// EVENT CODE //
	FB_AlarmCodeManager(
		bAlarm1			:= MesDataExd.AX_PowerCol[1].MesData.MesAcSwitchClosed,																							// AC Switch Closed for PCS 1
		bAlarm2			:= MesDataExd.MesData.MesOpened_Dc, 																											// DC Switch Closed
		bAlarm3			:= MesDataExd.MesData.OUT_CmdStandby, 																												// Soft stop command
		bAlarm4			:= MesDataExd.MesData.MesOnGrid,																													// OnGrid Mode is activated
		bAlarm5			:= MesDataExd.MesData.MesOffGrid, 																													// Offgrid Mode is activated
		bAlarm6			:= MesDataExd.MesData.OUT_CmdStart, 																												// Cmd Start
		bAlarm7			:= MesDataExd.MesData.OUT_CmdStop, 																												// Full stop command
		bAlarm8			:= MesDataExd.OUT_CmdBlackStart, 																											// Cmd BlackStart
		bAlarm9			:= MesDataExd.AX_PowerCol[1].MesRegAlarm2.9 OR MesDataExd.AX_PowerCol[2].MesRegAlarm2.9 OR MesDataExd.AX_PowerCol[3].MesRegAlarm2.9,			// Grid collapsed 
		bAlarm10		:= MesDataExd.AX_PowerCol[2].MesData.MesAcSwitchClosed,																							// AC Switch Closed for PCS 2
		bAlarm11		:= SEL(ParamNbPowerCol>2 ,  FALSE, MesDataExd.AX_PowerCol[3].MesData.MesAcSwitchClosed),																// AC Switch Closed for PCS 3
		bAlarm12		:= MesDataExd.MesData.MesOpened_Ac, 																											// Ac breaker is Closed. 
		bAlarm13		:= MesDataExd.MesData.MesState_Precharge,                                                                                            					// ESS - INV : Precharge
		bAlarm14		:= NOT MesDataExd.OUT_CmdGridMode,                                                                                                         // OnGrid command
		bAlarm15		:= MesDataExd.OUT_CmdGridMode, 																											// OffGrid command
		wAlarmCode		=>MesDataExd.MesData.MesEventCode);                                                                                           					// 
		

NumAlarmsActive := 0;
AX_AlarmWords := AX_AlarmWords_Null;
MesNbMots := 2;
FOR KK := 1 TO MesNbMots DO			// Combien j'ai de mots
	ID_Journal := 15 + (ParamEssNum-1) * MesNbMots * CstNbPcs_ESS_G + (ParamPcsNum - 1) * CstNbPcs_ESS_G + (KK- 1);
	FOR LL := 1 TO 15 DO 	// Les bits 
		WordTest := ROR(FUN_Alarms.AX_RecupWord[ID_Journal],LL);
		IF WordTest.0 THEN
			NumAlarmsActive := NumAlarmsActive + 1;
			AX_AlarmWords[NumAlarmsActive].Message := FUN_Alarms.AX_Journal[ID_Journal][LL].Message;
		ELSE
			AX_AlarmWords[NumAlarmsActive+1].Message := '';
		END_IF
	END_FOR
END_FOR		

NumAlarmsActiveJema := 0;
AX_AlarmWordsJema := AX_AlarmWordsJema_Null;
MesNbMots := 15;
FOR KK := 1 TO MesNbMots DO			// Combien j'ai de mots
	FOR LL := 1 TO 15 DO 	// Les bits 
		ID_Journal := 57 + (ParamEssNum-1) * MesNbMots * CstNbPcs_ESS_G + (ParamPcsNum - 1) * CstNbPcs_ESS_G + (KK- 1);
		WordTest := ROR(FUN_Alarms.AX_RecupWord[ID_Journal],LL);
		IF WordTest.0 THEN
			NumAlarmsActiveJema := NumAlarmsActiveJema + 1;
			AX_AlarmWordsJema[NumAlarmsActiveJema].Message := FUN_Alarms.AX_Journal[ID_Journal][LL].Message;
		ELSE
			AX_AlarmWordsJema[NumAlarmsActiveJema+1].Message := '';
		END_IF
	END_FOR
END_FOR
END_METHOD

METHOD M_CP
//////////////////
//  Emulator
/////////////////

VAR 
	// Method local variables (reinitialized at each cycle) 
	
END_VAR


SUPER^.M_CP() ; 




Trig_Cmd_Read(CLK:=IN_CmdToggleRead);
Trig_Cmd_Write(CLK:=IN_CmdToggleWrite);
	
IF Trig_Cmd_Read.Q THEN
	IN_CmdToggleRead := FALSE;
	MesDataExd.MesData.MesCP_Read := NOT MesDataExd.MesData.MesCP_Read;
END_IF


IF Trig_Cmd_Write.Q THEN
	IN_CmdToggleWrite := FALSE;
	MesDataExd.MesData.MesCP_Write := NOT MesDataExd.MesData.MesCP_Write;
END_IF
END_METHOD

METHOD M_Evaluate : BOOL
VAR_INPUT
END_VAR
VAR
	KK : UINT;
	bTest: BOOL;
	MesAlarmPcs: BOOL;
	AX_Journal : ARRAY[57..57] of array[1..15] of ST_ValuesAlarms;
END_VAR
// External values update :
//	DataSystemBMS 				:= AX_ESS[ParamEssNum].AX_Bat[ParamPcsNum].MesDataExd;

// Gestion des watchdogs
	Trig_Watchdog(CLK := MesHeartbeat_Old <> MesDataExd.MesData.MesHeartBeat);
	IF Trig_Watchdog.Q 	THEN
		MesHeartbeat_Old := MesDataExd.MesData.MesHeartBeat;
		MesStatusWatchdog := NOT MesStatusWatchdog;
	END_IF


// Gestion des Start/Stop par SOC Low

	TRIG_SocStop			(clk := NOT MesDataExd.MesData.MesState.0 AND NOT MesDataExd.MesData.MesState.4 AND DataSystemBMS.MesSoCConnected <= ParamSocStop);
	
	IF TRIG_SocStop.Q THEN
		MesDataExd.MesData.MesState.4 := TRUE;
	END_IF
	
	
	TRIG_SocStop_Again(CLK := Time_Discharge_LowSoc > ParamTimeLowSocToRecharge);
	IF NOT MesDataExd.MesData.MesState.0 AND MesDataExd.MesData.MesState.4 AND MesDataExd.MesData.MesPdc >= 0 THEN
		Time_Discharge_LowSoc := Time_Discharge_LowSoc + TIME() - Time_Start_Discharge_LowSoc;
	ELSIF MesDataExd.MesData.MesState.0 AND (NOT MesDataExd.MesData.MesState.4 OR Time_Discharge_LowSoc >= ParamTimeLowSocToRecharge) THEN
		Time_Discharge_LowSoc := T#0S;
	END_IF
	Time_Start_Discharge_LowSoc := TIME();
	
	TRIG_BackToNormalSoc(CLK := MesDataExd.MesData.MesState.4 AND DataSystemBMS.MesSoCConnected > ParamSocStop);
	IF TRIG_BackToNormalSoc.Q THEN
		MesDataExd.MesData.MesState.4 := 0;
	END_IF
	
	
	
	IF ParamAllowRechargeLowSoc THEN
		TRIG_Recharge_LowSoc(CLK := NOT MesDataExd.MesData.MesState.0 AND NOT MesDataExd.MesData.MesState.4 AND DataSystemBMS.MesSoCConnected <= ParamSocRecharge);
		IF TRIG_Recharge_LowSoc.Q THEN
			MesDataExd.MesData.MesState.3 := TRUE;
		END_IF
		
		TRIG_RechargeBackToNormalSoc(CLK := MesDataexd.MesData.MesState.3 AND DataSystemBMS.MesSoCConnected >= ParamSocMin_G);
		IF TRIG_RechargeBackToNormalSoc.Q THEN
			MesDataexd.MesData.MesState.3 := FALSE;
		END_IF
	END_IF
	
	
	
// PROPERTIES UPDATE // 
	// Controller
	
	MesDataExd.MesData.MesP 	:= 0 ; 
	MesDataExd.MesData.MesPdc 	:= 0 ;
	MesDataExd.MesData.MesQ 	:= 0 ; 
	MesDataExd.MesData.MesI 	:= 0 ; 			
	MesDataExd.MesData.MesIdc 	:= 0 ; 		
	MesDataExd.MesData.MesTemp	:= 0 ;
	
	MesDataExd.MesData.MesAlarmCom					:= TRUE ; 	// All PCS in Com alarm . 			
	MesDataExd.MesData.MesALOPowerCol_Connected 			:= FALSE; 	// At least one inverter connected and not in alarm			
	MesDataExd.MesData.MesFreqReg_Active 			:= FALSE;
	MesDataExd.MesData.MesUReg_Active 				:= FALSE;

	// Update PCS Values	
	FOR KK:= 1 TO ParamNbPowerCol DO 
		MesDataExd.MesData.MesP 						:= MesDataExd.AX_PowerCol[KK].MesData.MesP + MesDataExd.MesData.MesP  ; 
		MesDataExd.MesData.MesI 						:= MesDataExd.AX_PowerCol[KK].MesData.MesI + MesDataExd.MesData.MesI  ; 
		MesDataExd.MesData.MesPdc 						:= MesDataExd.AX_PowerCol[KK].MesData.MesPdc + MesDataExd.MesData.MesPdc  ; 
		MesDataExd.MesData.MesQ 						:= -MesDataExd.AX_PowerCol[KK].MesData.MesQ + MesDataExd.MesData.MesQ  ; 
		MesDataExd.MesData.MesIdc 						:= MesDataExd.AX_PowerCol[KK].MesData.MesIdc + MesDataExd.MesData.MesIdc  ; 
		MesDataExd.MesData.MesFreqReg_Active			:= MesDataExd.MesData.MesFreqReg_Active 			OR MesDataExd.AX_PowerCol[KK].MesDeratingWord.6 OR MesDataExd.AX_PowerCol[KK].MesDeratingWord.7 ;
		MesDataExd.MesData.MesUReg_Active				:= MesDataExd.MesData.MesUReg_Active 				OR MesDataExd.AX_PowerCol[KK].MesDeratingWord.4 OR MesDataExd.AX_PowerCol[KK].MesDeratingWord.5 ;
		MesAlarmPcs										:= MesDataExd.AX_PowerCol[KK].MesRegAlarm0 > 0 		OR MesDataExd.AX_PowerCol[KK].MesRegAlarm1 > 0 	OR MesDataExd.AX_PowerCol[KK].MesRegAlarm2 > 0 OR MesDataExd.AX_PowerCol[KK].MesRegAlarm3 > 0 OR MesDataExd.AX_PowerCol[KK].MesRegAlarm4 > 0;                                        	
		MesDataExd.MesData.MesAlarmCom					:= MesDataExd.MesData.MesAlarmCom 					AND AX_PcsHeartbit[KK];
		MesDataExd.MesData.MesALOPowerCol_Connected 			:= MesDataExd.MesData.MesALOPowerCol_Connected 			OR MesDataExd.AX_PowerCol[KK].MesData.MesAcSwitchClosed (*FAT TESTAND NOT MesAlarmPcs *);
	
		MesDataExd.MesData.MesTemp 						:= MesDataExd.MesData.MesTemp + MesDataExd.AX_PowerCol[KK].MesData.MesTemp/ParamNbPowerCol;
	
			
	END_FOR 
	
	MesDataExd.MesData.MesCosPhi 				:= SEL(	(MesDataExd.MesData.MesP=0) AND  (MesDataExd.MesData.MesQ =0 ), MesDataExd.MesData.MesP / SQRT(EXPT(MesDataExd.MesData.MesP, 2) + EXPT(MesDataExd.MesData.MesQ, 2))   , 1) ; 		
	MesDataExd.MesData.MesFreq					:= SEL(MesDataExd.AX_PowerCol[1].MesData.MesFreq=0 ,MesDataExd.AX_PowerCol[1].MesData.MesFreq , SEL(MesDataExd.AX_PowerCol[2].MesData.MesFreq=0 ,MesDataExd.AX_PowerCol[2].MesData.MesFreq ,MesDataExd.AX_PowerCol[3].MesData.MesFreq ))   ; 		
	MesDataExd.MesData.MesU 					:= SEL(MesDataExd.AX_PowerCol[1].MesData.MesU=0 ,MesDataExd.AX_PowerCol[1].MesData.MesU , SEL(MesDataExd.AX_PowerCol[2].MesData.MesU=0 ,MesDataExd.AX_PowerCol[2].MesData.MesU ,MesDataExd.AX_PowerCol[3].MesData.MesU ))   ; 		
	MesDataExd.MesData.MesUdc 					:= SEL(MesDataExd.AX_PowerCol[1].MesData.MesUdc=0 ,MesDataExd.AX_PowerCol[1].MesData.MesUdc , SEL(MesDataExd.AX_PowerCol[2].MesData.MesUdc=0 ,MesDataExd.AX_PowerCol[2].MesData.MesUdc ,MesDataExd.AX_PowerCol[3].MesData.MesUdc ))   ; 			
	 
	
//--------------------------------------------------------------------------------//
// 							Gestion des setpoints								  //
//--------------------------------------------------------------------------------//
	
// Gestion de la puissance dispo batterie		
	//  MesDataExd.MesData.CalDynamicEfficiencyPcs := (ParamRendementPcsNom  - ParamRendementPcsMin)* (1-EXP(-(abs.MesDataExd.MesData.CalP)/ParamPnom)*100/ParamTauxDeChargeRef)) + ParamRendementPcsMin;

// Gestion des limites hautes de SoC
	RS_hystlimitmax(SET:= DataSystemBMS.MesSoCConnected >= ParamSocMax_G , RESET1:= DataSystemBMS.MesSoCConnected < ParamSocHigh) ; 
	RS_hystlimitmin(SET:= DataSystemBMS.MesSoCConnected <= ParamSocMin_G , RESET1:= DataSystemBMS.MesSoCConnected > ParamSocLow) ; 
	
	IF DataSystemBMS.MesSoCConnected >= ParamSocHigh THEN
		CalPmaxCorr_highSoC := (ParamSocMax_G - DataSystemBMS.MesSoCConnected)/(ParamSocMax_G - ParamSocHigh );
	ELSE 
		CalPmaxCorr_highSoC := 1 ;
	END_IF 
	IF DataSystemBMS.MesSoCConnected <= ParamSocLow THEN
		CalPminCorr_lowSoC := (ParamSocMin_G - DataSystemBMS.MesSoCConnected)/(ParamSocMin_G - ParamSocLow );
	ELSE
		CalPminCorr_lowSoC := 1;
	END_IF
	
	IF (datasystembms.MesData.MesCCL <> 0 OR datasystembms.MesData.MesDCL <> 0) AND DataSystemBMS.MesUdcConnected <> 0 THEN
		MesDataExd.MesData.MesSmax_ChargeFromBat 		:=  SEL(RS_hystlimitmax.Q1, 1, 0) * CalPmaxCorr_highSoC * MIN(DataSystemBMS.MesData.MesCCL*ParamChargeEfficiency/100,	ParamPn);
		MesDataExd.MesData.MesSmax_DischargeFromBat 	:=  SEL(RS_hystlimitmin.Q1, 1, 0) * CalPminCorr_lowSoC * MIN(DataSystemBMS.MesData.MesDCL*ParamDischargeEfficiency/100,	ParamPn);
	ELSE
		MesDataExd.MesData.MesSmax_ChargeFromBat := 0;
		MesDataExd.MesData.MesSmax_DischargeFromBat := 0;
	END_IF
	

// Local
	// Si je suis en local, je désactive le micro cycling et je réecris le setpoint d'input	
		IF MesDataExd.MesData.OUT_CmdPcsLocal THEN
			IN_SetptP := IN_SetptP_Local;
			IN_SetptQ := IN_SetptQ_Local;
			IN_SetptU := IN_SetptU_Local;
			IN_SetptF := IN_SetptF_Local;
		END_IF

	MesDataExd.MesData.OUT_SetptSMax := MIN(MesDataExd.MesData.MesAvailability * MesDataExd.MesData.MesSnom/100.0,  ParamPn);

IF ParamPoverQ THEN 
	// Le setpoint Max correspond à la dispo * la puissance nominale
	MesDataExd.MesData.OUT_SetptPMax := MIN(MesDataExd.MesData.MesSmax_DischargeFromBat, MesDataExd.MesData.OUT_SetptSMax);
	MesDataExd.MesData.OUT_SetptPMin := - MIN(MesDataExd.MesData.MesSmax_ChargeFromBat, MesDataExd.MesData.OUT_SetptSMax);

	// Min
	IF ABS(MesDataExd.MesData.OUT_SetptSMax) > ABS(MesDataExd.MesData.OUT_SetptP) THEN
		MesDataExd.MesData.OUT_SetptQMax		:= MIN(ParamQn, SQRT(EXPT(MesDataExd.MesData.OUT_SetptSMax, 2) - EXPT(MesDataExd.MesData.OUT_SetptP, 2)));
	ELSE
		MesDataExd.MesData.OUT_SetptQMax := 0;
	END_IF
	IF ABS(MesDataExd.MesData.OUT_SetptSMax) > ABS(MesDataExd.MesData.OUT_SetptP) THEN
		MesDataExd.MesData.OUT_SetptQMin		:= -MIN(ParamQn,SQRT( EXPT(MesDataExd.MesData.OUT_SetptSMax, 2) - EXPT(MesDataExd.MesData.OUT_SetptP, 2)));
	ELSE 
		MesDataExd.MesData.OUT_SetptQMin := 0;
	END_IF
ELSE
	MesDataExd.MesData.OUT_SetptQMax := SEL(MesDataExd.MesData.MesP = 0, SEL(MesDataExd.MesData.MesP>0, MesDataExd.MesData.MesSmax_ChargeFromBat, MesDataExd.MesData.MesSmax_DischargeFromBat), MIN(MesDataExd.MesData.MesSmax_ChargeFromBat, MesDataExd.MesData.MesSmax_DischargeFromBat));
	MesDataExd.MesData.OUT_SetptQMin := -MesDataExd.MesData.OUT_SetptQMax;
		
	MesDataExd.MesData.OUT_SetptPMax		:= MIN(SQRT(EXPT(MesDataExd.MesData.MesSmax_ChargeFromBat, 2) - EXPT(MesDataExd.MesData.OUT_SetptQ, 2)),  SEL(DataSystemBMS.MesSoCConnected < ParamSocMin_G, ParamPn, 0));
	MesDataExd.MesData.OUT_SetptPMin		:= MAX(SQRT(EXPT(MesDataExd.MesData.MesSmax_DischargeFromBat, 2) - EXPT(MesDataExd.MesData.OUT_SetptQ, 2)),  SEL(DataSystemBMS.MesSoCConnected > ParamSocMax_G, ParamPn, 0));
END_IF

// J'affecte les variables que je vais écrire
IF MesDataExd.OUT_CmdP THEN
	IF ParamAllowRechargeLowSoc AND MesDataExd.MesData.MesState.3 THEN
		IN_SetptP := MIN(IN_SetptP, - ABS(ParamPrechargeLowSoc)) ;
	END_IF
	MesDataExd.MesData.OUT_SetptP		:= MIN(MAX(IN_SetptP, MesDataExd.MesData.OUT_SetptPMin), MesDataExd.MesData.OUT_SetptPMax);
	
ELSE
	MesDataExd.MesData.OUT_SetptP 		:= 0;
END_IF

IF MesDataExd.OUT_CmdQ THEN
	MesDataExd.MesData.OUT_SetptQ		:= -MIN(MAX(IN_SetptQ, MesDataExd.MesData.OUT_SetptQMin), MesDataExd.MesData.OUT_SetptQMax);
ELSE
	MesDataExd.MesData.OUT_SetptQ 		:= 0;
END_IF

MesDataExd.OUT_SetptV := IN_SetptU;
MesDataExd.OUT_SetptF := IN_SetptF;


TON_CmdQ_On				(IN := MesDataExd.OUT_CmdQ 						AND NOT MesDataExd.MesData.MesID_State_Inv.4, PT := ParamTimeoutCmdQ);		
TON_CmdQ_Off			(IN :=  NOT MesDataExd.OUT_CmdQ  				AND MesDataExd.MesData.MesID_State_Inv.4, PT := ParamTimeoutCmdQ);				   	
TON_CmdCosPhi_On		(IN := MesDataExd.OUT_CmdCosPhi 				AND NOT MesDataExd.MesData.MesID_State_Inv.5, PT := ParamTimeoutCmdCosPhi);		
TON_CmdCosPhi_Off		(IN :=  NOT MesDataExd.OUT_CmdCosPhi 			AND MesDataExd.MesData.MesID_State_Inv.5, PT := ParamTimeoutCmdCosPhi);		
TON_FreqReg_On			(IN := MesDataExd.OUT_CmdFreqregMode 			AND NOT MesDataExd.MesData.MesID_State_Inv.2, PT := ParamTimeoutPvF);			
TON_FreqReg_Off			(IN :=  NOT MesDataExd.OUT_CmdFreqregMode 		AND MesDataExd.MesData.MesID_State_Inv.2, PT := ParamTimeoutPvF	);		
TON_UReg_On				(IN := MesDataExd.OUT_CmdUregMode 				AND NOT MesDataExd.MesData.MesID_State_Inv.1, PT := ParamTimeoutQvU	);		
TON_UReg_Off			(IN :=  NOT MesDataExd.OUT_CmdUregMode 			AND MesDataExd.MesData.MesID_State_Inv.1, PT := ParamTimeoutQvU	);		
TON_CmdGridFormer		(IN := MesDataExd.OUT_CmdGridMode 				AND NOT MesDataExd.MesData.MesID_State_Inv.10, PT := ParamTimeoutGridFormerTransition	);		
TON_CmdGridFeeder		(IN :=  NOT MesDataExd.OUT_CmdGridMode			AND MesDataExd.MesData.MesID_State_Inv.10, PT := ParamTimeoutGridFeederTransition	);		
TON_CmdStop				(IN := MesDataExd.MesData.OUT_CmdStop					AND MesDataExd.MesData.MesState.0);
TON_CmdStart			(IN := MesDataExd.MesData.OUT_CmdStart					AND NOT MesDataExd.MesData.MesState.0);
END_METHOD

METHOD M_Init

VAR 

END_VAR
SUPER^.M_Init() ; 

MesDataExd.MesData.MesState.0 := TRUE; // Initialize state to OFF

MesDataExd.OUT_CmdP := TRUE;
MesDataExd.OUT_CmdQ := TRUE;

MesDataExd.MesData.MesCP_Read := TRUE;
MesDataExd.MesData.MesCP_Write := TRUE;
END_METHOD

METHOD M_Read
//////////////////
//  Read Modbus Variable for PCS . 
/////////////////

VAR 
	// Method local variables (reinitialized at each cycle) 
	MW 						: FB_MergeWordsToDint; 

	
	MesPsetPt_Temp 			: REAL ;
	MesQsetPt_Temp			: REAL ;
	MesPavailablePcs_Temp	: REAL;
	MesPavailable_Temp		: REAL;
	
	ComErrorPcs_Temp		: WORD;
	
	KK						: BYTE;  					// FOR Loop 
	LL						: BYTE;						// Alarm Loop

	MesPsetPtPcs_temp		: ARRAY[1..CstNbPcs_ESS_G] OF  REAL; // Setpt lu sur le module
	MesQsetPtPcs_temp		: ARRAY[1..CstNbPcs_ESS_G] OF  REAL;

	AX_Qty					: ARRAY[1..3] OF WORD := [75, 68, 68];
	AX_Addr					: ARRAY[1..3] OF WORD := [1100, 1200, 1300];
	bReadChanged : BOOL;

END_VAR


IF MesDataExd.MesData.MesCP_Read  THEN	
// MODBUS REQUEST//

		ModbusRead[4]
		(
			tTimeout		:= ParamTimeout,
			nUnitID			:= ParamUnitID,
			sIPAddr			:= ParamIPAddress ,
			ClockRead		:= ClockRead AND MesDataExd.MesData.MesCP_Read,
			nTcpPort		:= ParamTcpPort,
			nQuantity		:= 75,
			Reset			:= IN_CmdReset,
			nMBAddr			:= 1100  ,//Access every PCS power modules
			cbLength		:= SIZEOF(MesBlock1_Temp[4]) , 
			pDestAddr		:= ADR(MesBlock1_Temp[4]),
			ModbusReadAlarm	=>MesModbusReadAlarm[4]
		);
			
	bReadChanged := MEMCMP(pBuf1 := ADR(MesBlock1_Temp_Old), pBuf2 := ADR(MesBlock1_Temp), n := SIZEOF(MesBlock1_Temp))<> 0;
	
	IF bReadChanged THEN
		MEMCPY(destAddr := ADR(MesBlock1_Temp_Old), srcAddr := ADR(MesBlock1_Temp), n := SIZEOF(MesBlock1_Temp_Old));
	END_IF
	TP_ReadCompleted(IN := bReadChanged, pt := ParamClockReadTime/2, Q=>MesDataExd.MesReadCompleted);

			
	// MODBUS REQUEST//
		FOR KK:=1 TO ParamNbPowerCol DO 	
			ModbusRead[KK]
			(
				tTimeout		:= ParamTimeout,
				nUnitID			:= ParamUnitID,
				sIPAddr			:= ParamIPAddress,
				ClockRead		:= ClockRead AND MesDataExd.MesData.MesCP_Read,
				nTcpPort		:= ParamTcpPort,
				nQuantity		:= AX_Qty[KK],
				Reset			:= IN_CmdReset,
				nMBAddr			:= AX_Addr[KK] ,
				cbLength		:= SIZEOF(MesBlock1_Temp[KK]) , 
				pDestAddr		:= ADR(MesBlock1_Temp[KK]),
				ModbusReadAlarm	=>MesModbusReadAlarm[KK]
			);
		END_FOR
		
		
	// MODBUS BLOCK SEPARATION/
		// Block1 (PCS) 
		FOR KK:=1 TO ParamNbPowerCol DO 	// Value per Power Column (3 per inverter IBX3)
			// Measurements
			MW( WORD_STRONG:= MesBlock1_Temp[KK][1], SIGNED:=TRUE, FIX:=1 , SIZE:=1, VAR_OUT := MesDataExd.AX_PowerCol[KK].MesData.MesUdc); 
			MW( WORD_STRONG:= MesBlock1_Temp[KK][2], SIGNED:=TRUE, FIX:=1 , SIZE:=1, VAR_OUT := MesDataExd.AX_PowerCol[KK].MesData.MesIdc); //Vérifier les signes
			MW( WORD_STRONG:= MesBlock1_Temp[KK][3], SIGNED:=FALSE, FIX:=1 , SIZE:=1, VAR_OUT := MesDataExd.AX_PowerCol[KK].MesData.MesU);
			MW( WORD_STRONG:= MesBlock1_Temp[KK][6], SIGNED:=FALSE, FIX:=1 , SIZE:=1, VAR_OUT := MesDataExd.AX_PowerCol[KK].MesData.MesI1); //Vérifier les signes
			MW( WORD_STRONG:= MesBlock1_Temp[KK][7], SIGNED:=FALSE, FIX:=1 , SIZE:=1, VAR_OUT := MesDataExd.AX_PowerCol[KK].MesData.MesI2); //Vérifier les signes
			MW( WORD_STRONG:= MesBlock1_Temp[KK][8], SIGNED:=FALSE, FIX:=1 , SIZE:=1, VAR_OUT := MesDataExd.AX_PowerCol[KK].MesData.MesI3); //Vérifier les signes
			MW( WORD_STRONG:= MesBlock1_Temp[KK][9], SIGNED:=TRUE, FIX:=1 , SIZE:=1, VAR_OUT := MesDataExd.AX_PowerCol[KK].MesData.MesPdc); // Vérifier les signes
			MW( WORD_STRONG:= MesBlock1_Temp[KK][10], SIGNED:=TRUE, FIX:=1 , SIZE:=1, VAR_OUT := MesDataExd.AX_PowerCol[KK].MesData.MesP); // Vérifier les signes
			MW( WORD_STRONG:= MesBlock1_Temp[KK][11], SIGNED:=TRUE, FIX:=1 , SIZE:=1, VAR_OUT := MesDataExd.AX_PowerCol[KK].MesData.MesQ);// Vérifier les signes
			MW( WORD_STRONG:= MesBlock1_Temp[KK][12], SIGNED:=FALSE, FIX:=3 , SIZE:=1, VAR_OUT := MesDataExd.AX_PowerCol[KK].MesData.MesCosPhi);
			MW( WORD_STRONG:= MesBlock1_Temp[KK][13], SIGNED:=FALSE, FIX:=2 , SIZE:=1, VAR_OUT := MesDataExd.AX_PowerCol[KK].MesData.MesFreq);
			
			// Inputs (Temp and IO)
			MW( WORD_STRONG:= MesBlock1_Temp[KK][15], SIGNED:=TRUE, FIX:=1 , SIZE:=1, VAR_OUT := MesDataExd.AX_PowerCol[KK].MesTempControl);
			MW( WORD_STRONG:= MesBlock1_Temp[KK][18], SIGNED:=TRUE, FIX:=1 , SIZE:=1, VAR_OUT := MesDataExd.AX_PowerCol[KK].MesTempPowerUnit);
	
			// Alarms
		MesDataExd.AX_PowerCol[KK].MesRegAlarm0:=MesBlock1_Temp[KK][24];
		MesDataExd.AX_PowerCol[KK].MesRegAlarm1:=MesBlock1_Temp[KK][25];
		MesDataExd.AX_PowerCol[KK].MesRegAlarm2:=MesBlock1_Temp[KK][26];
		MesDataExd.AX_PowerCol[KK].MesRegAlarm3:=MesBlock1_Temp[KK][27];
		MesDataExd.AX_PowerCol[KK].MesRegAlarm4:=MesBlock1_Temp[KK][28];					
	
			MW( WORD_STRONG:= MesBlock1_Temp[KK][48], SIGNED:=TRUE, FIX:=1 , SIZE:=1, VAR_OUT := MesDataExd.AX_PowerCol[KK].MesTempCabinet);
			
			// States
		MesDataExd.AX_PowerCol[KK].MesData.MesAcSwitchClosed := MesBlock1_Temp[KK][61].2 ;	// AC contactor status
		MesDataExd.AX_PowerCol[KK].MesDoorOpened := NOT MesBlock1_Temp[KK][61].6; // Door : 1= Close, O= Open
		MesDataExd.AX_PowerCol[KK].MesDeratingWord := MesBlock1_Temp[KK][62] ;
			
			MW( WORD_STRONG:= MesBlock1_Temp[KK][68], SIGNED:=FALSE, FIX:=0 , SIZE:=1, VAR_OUT := MesDataExd.AX_PowerCol[KK].MesHeartbit);
			
	
		END_FOR
	
		// Inverter states (à tester)
	
	MesDataExd.MesData.MesID_State_Inv				:= MesBlock1_Temp[4][67];
	MesDataExd.MesData.MesSnom						:= MIN(WORD_TO_REAL(MesBlock1_Temp[1][69]),ParamSn);	
	MesDataExd.MesData.MesAvailability				:= WORD_TO_REAL(MesBlock1_Temp[4][70]);
		
	MW( WORD_STRONG := MesBlock1_Temp[4][71], SIZE := 1, FIX := 0, SIGNED := FALSE, VAR_OUT := MesDataExd.MesHumidity);
	MW( WORD_STRONG := MesBlock1_Temp[4][72], SIZE := 1, FIX := 1, SIGNED := TRUE, VAR_OUT := MesDataExd.MesData.MesTemp);
	MesDataExd.MesData.MesTemp 						:= WORD_TO_REAL(MesBlock1_Temp[4][72])/10;
	MesDataExd.MesData.MesState_Precharge 			:= WORD_TO_BOOL(MesBlock1_Temp[4][73]);
	MesDataExd.MesData.MesOpened_Dc					:= NOT MesBlock1_Temp[4][74].0;
	MesDataExd.MesData.MesOpened_Ac					:= NOT  MesBlock1_Temp[4][61].0;
	MesDataExd.MesState_SoCLimitReached				:= MesBlock1_Temp[4][74].2;
	MesDataExd.MesData.MesOffGrid					:= MesBlock1_Temp[4][74].3;
	MesDataExd.MesData.MesOnGrid					:= MesBlock1_Temp[4][74].4;
	MesDataExd.MesData.MesHeartBeat					:= MesBlock1_Temp[4][75];
	
	
	
	
	
END_IF
END_METHOD

METHOD M_StateManager
//////////////////
// Detect which is the state of the PCS system . 
/////////////////

VAR 
	// Method local variables (reinitialized at each cycle) 

	
	ELS: INT;
END_VAR


MesDataExd.MesData.MesState.0 	:= 0;
IF NOT MesDataExd.MesData.MesALOPowerCol_Connected OR MesDataExd.MesData.MesOpened_Ac OR  MesDataExd.MesData.MesOpened_Dc THEN 
	// OFF State :  No Charger connected or all charger in alarm
	MesDataExd.MesData.MesState.0 	:= 1 ; 
END_IF

MesDataExd.MesData.MesState.1 	:= 0 ; 
IF MesDataExd.MesData.MesOffGrid THEN
	// Feeding master
	MesDataExd.MesData.MesState.1 	:= 1 ; 
END_IF	

MesDataExd.MesData.MesState.2 	:= 0 ; 
IF MesDataExd.MesData.OUT_CmdPcsLocal THEN
	MesDataExd.MesData.MesState.2 	:= 1 ; 
END_IF




SUPER^.M_StateManager() ;
END_METHOD

METHOD M_WriteCommand
//////////////////
//  Modbus Write of the command for the PCS. 
/////////////////

VAR 
	// Method local variables (reinitialized at each cycle) 
	
	AX_Adr			: ARRAY[1..3] OF UINT := [1707	, 1802	, 	0217	];
	AX_QTY			: ARRAY[1..3] OF BYTE := [41	, 33	, 	2		];
	AX_UnitID		: ARRAY[1..3] OF BYTE := [1		, 1		, 	1		];	

	KK: INT;
	
END_VAR
TRIG_CmdP_On			(CLK := IN_CmdP_On);						
TRIG_CmdP_Off			(CLK := IN_CmdP_Off);							
TRIG_CmdQ_On			(CLK := IN_CmdQ_On);                        
TRIG_CmdQ_Off			(CLK := IN_CmdQ_Off);                      
TRIG_CmdCosPhi_On		(CLK := IN_CmdCosPhi_On);              
TRIG_CmdCosPhi_Off		(CLK := IN_CmdCosPhi_Off);            
TRIG_CmdReset			(CLK := IN_CmdReset);
TRIG_FreqReg_On			(CLK := IN_CmdFreqregOn);
TRIG_FreqReg_Off		(CLK := IN_CmdFreqregOff);
TRIG_UReg_On			(CLK := IN_CmdUregOn);			
TRIG_UReg_Off			(CLK := IN_CmdUregOff);
TRIG_CmdGridFormer		(CLK := IN_CmdGridFormer);
TRIG_CmdGridFeeder		(CLK := IN_CmdGridFeeder);
TRIG_CmdOpenAC			(CLK := IN_CmdOpenAC);
TRIG_CmdOpenDC			(CLk := IN_CmdOpenDC);
TRIG_CmdStop			(CLK := IN_CmdStop);
TRIG_CmdStandby			(CLK := (IN_CmdStandby OR TON_BatComAlarm.Q)  AND NOT TP_CmdStop.Q );
TRIG_CmdStart			(CLK := IN_CmdStart AND NOT TP_CmdStop.Q AND NOT IN_CmdStopOperation AND (NOT IN_CmdPreventStart OR MesDataExd.MesData.OUT_CmdPcsLocal));
TRIG_CmdBlackStart		(CLK := IN_CmdBlackStart);	


TP_CmdPreStop			(IN := TRIG_CmdStop.Q, 																		PT := T#1S500MS);
TP_CmdPreStart			(IN := TRIG_CmdStart.Q, 																	PT := ParamTimePulseTrig);
TP_CmdOpenAC			(IN := TRIG_CmdOpenAC.Q, 																	PT := ParamTimePulseTrig);
TP_CmdOpenDC			(IN := TRIG_CmdOpenDC.Q, 																	PT := ParamTimePulseTrig);
TP_CmdStop				(IN := F_TrigPreStop.Q, 																	PT := ParamTimePulseTrig);
TP_CmdStart				(IN := F_TrigPreStart.Q, 																	PT := ParamTimePulseTrig);
TP_CmdStandby			(IN := TRIG_CmdStop.Q OR TRIG_CmdStandby.Q OR TRIG_SocStop.Q OR TRIG_SocStop_Again.Q, 	PT := ParamTimePulseTrig);
TP_Reset				(IN := TRIG_CmdReset.Q, 																	PT := ParamTimePulseTrig);
                		
                		
F_TrigPreStart			(CLK := TP_CmdPreStart.Q);
F_TrigPreStop			(CLK := TP_CmdPreStop.Q);


IF TRIG_CmdBlackStart.Q THEN
	IN_CmdBlackStart := FALSE;
END_IF
IF TRIG_CmdStop.Q THEN
	IN_CmdStop := FALSE;
END_IF
IF TRIG_CmdStart.Q THEN
	AX_ESS[ParamEssNum].AX_BAT[ParamPcsNum].IN_CmdCloseDC := TRUE;
	IN_CmdStart := FALSE;
END_IF
IF TRIG_CmdStandby.Q THEN
	IN_CmdStandby := FALSE;
END_IF

IF TRIG_CmdReset.Q THEN
	IN_CmdReset := FALSE;
END_IF

IF TRIG_CmdP_Off.Q THEN
	MesDataExd.OUT_CmdP := FALSE;
	IN_CmdP_Off := FALSE;
END_IF

IF TRIG_CmdP_On.Q THEN
	MesDataExd.OUT_CmdP := TRUE;
	IN_CmdP_On := FALSE;
END_IF
IF TRIG_CmdQ_Off.Q OR TRIG_CmdCosPhi_On.Q THEN
	MesDataExd.OUT_CmdQ := FALSE;
	IN_CmdQ_Off := FALSE;
END_IF
IF TRIG_CmdQ_On.Q THEN
	MesDataExd.OUT_CmdQ := TRUE;
	IN_CmdQ_On := FALSE;
END_IF

IF TRIG_CmdCosPhi_Off.Q OR TRIG_CmdQ_On.Q THEN
	MesDataExd.OUT_CmdCosPhi := FALSE;
	IN_CmdCosPhi_Off := FALSE;
END_IF

IF TRIG_CmdCosPhi_On.Q THEN
	MesDataExd.OUT_CmdCosPhi := TRUE;
	MesDataExd.OUT_SetptCosPhi	:= IN_SetptCosPhi;
	IN_CmdCosPhi_On := FALSE;
END_IF

IF TRIG_FreqReg_On.Q THEN
	MesDataExd.OUT_CmdFreqregMode := TRUE;
	IN_CmdFreqregOn := FALSE;
END_IF
IF TRIG_FreqReg_Off.Q THEN
	MesDataExd.OUT_CmdFreqregMode := FALSE;
	IN_CmdFreqregOff := FALSE;
END_IF

IF TRIG_UReg_On.Q THEN
	MesDataExd.OUT_CmdUregMode := TRUE;
	IN_CmdUregOn := FALSE;
END_IF
IF TRIG_UReg_Off.Q THEN
	MesDataExd.OUT_CmdUregMode := FALSE;
	IN_CmdUregOff := FALSE;
END_IF
	
IF TRIG_CmdGridFormer.Q THEN
	MesDataExd.OUT_CmdGridMode := TRUE;
	IN_CmdGridFormer := FALSE;
END_IF 
IF TRIG_CmdGridFeeder.Q OR TRIG_CmdStop.Q THEN //Si on fait une commande stop, on passe le mode en grid feeder
	MesDataExd.OUT_CmdGridMode := FALSE;
	IN_CmdGridFeeder := FALSE;
END_IF


IF IN_CmdPcsLocal THEN
	IN_CmdPcsLocal := FALSE;
	MesDataExd.MesData.OUT_CmdPcsLocal := NOT MesDataExd.MesData.OUT_CmdPcsLocal;
END_IF

IN_CmdWatchdog := CalLocalTimeStruct.wSecond MOD 2 = 0;

MesDataExd.MesData.OUT_CmdStop 			:= TP_CmdStop.Q;
MesDataExd.MesData.OUT_CmdStart 		:= TP_CmdStart.Q;
MesDataExd.OUT_CmdBlackStart 	:= TP_CmdBlackStart.Q;
MesDataExd.MesData.OUT_CmdStandby 		:= TP_CmdStandby.Q;


Trig_Write[1](CLK := MEMCMP(pBuf1 :=ADR(AX_Cmd[1]), pBuf2 := ADR(AX_Cmd_Old[1]), n := SIZEOF(AX_CMD[1]))<>0);
Trig_Write[2](CLK := MEMCMP(pBuf1 :=ADR(AX_Cmd[2]), pBuf2 := ADR(AX_Cmd_Old[2]), n := SIZEOF(AX_CMD[2]))<>0);
Trig_Write[3](CLK := MEMCMP(pBuf1 :=ADR(AX_Cmd[3]), pBuf2 := ADR(AX_Cmd_Old[3]), n := SIZEOF(AX_CMD[3]))<>0);

IF MEMCMP(pBuf1 :=ADR(AX_Cmd[1]), pBuf2 := ADR(AX_Cmd_Old[1]), n := SIZEOF(AX_CMD[1]))<>0 THEN
	MEMCPY(destAddr := ADR(AX_Cmd_Old[1]), srcAddr := ADR(AX_Cmd[1]), n:= SIZEOF(AX_Cmd[1]));
END_IF
IF MEMCMP(pBuf1 :=ADR(AX_Cmd[2]), pBuf2 := ADR(AX_Cmd_Old[2]), n := SIZEOF(AX_CMD[2]))<>0 THEN
	MEMCPY(destAddr := ADR(AX_Cmd_Old[2]), srcAddr := ADR(AX_Cmd[2]), n:= SIZEOF(AX_Cmd[2]));
END_IF		
IF MEMCMP(pBuf1 :=ADR(AX_Cmd[3]), pBuf2 := ADR(AX_Cmd_Old[3]), n := SIZEOF(AX_CMD[3]))<>0 THEN
	MEMCPY(destAddr := ADR(AX_Cmd_Old[3]), srcAddr := ADR(AX_Cmd[3]), n:= SIZEOF(AX_Cmd[3]));
END_IF			

	// Manouvers (41708)
		AX_Cmd[1][1].1:= IN_CmdOpenAC;
		AX_Cmd[1][1].2:= IN_CmdOpenDC;
		
	// SoC	
		AX_Cmd[1][2]  := REAL_TO_WORD(ParamFreqRegSoCmax); 
		AX_Cmd[1][3]  := REAL_TO_WORD(ParamFreqRegSoCmin); 
		AX_Cmd[1][4]  := REAL_TO_WORD(TRUNC(DataSystemBMS.MesSoCConnected));		// SoC connected 
		
		
	// Param voltage regulation (activate in Function Mode)
		// Regulation from voltage
		AX_Cmd[1][7]  := REAL_TO_WORD(ParamQfU_UDbHigh)		; 
		AX_Cmd[1][8]  := REAL_TO_WORD(ParamQfU_Umax)		  	; 
		AX_Cmd[1][9]  := REAL_TO_WORD(ParamQfU_UDbLow)	 	; 
		AX_Cmd[1][10] := REAL_TO_WORD( ParamQfU_Umin	)  		; 
		
		IF ParamNbPowerCol > 0 THEN 
			AX_Cmd[1][11]  := REAL_TO_WORD(MIN(MAX(-ParamQfU_QDbHigh*ParamNbPowerCol/ParamPn*1000.0, -1000 ), 1000))			; 
			AX_Cmd[1][12]  := REAL_TO_WORD(MIN(MAX(-ParamQfU_Qmax*ParamNbPowerCol/ParamPn*1000.0, -1000 ), 1000))			  	; 
			AX_Cmd[1][13]  := REAL_TO_WORD(MIN(MAX(-ParamQfU_QDbLow*ParamNbPowerCol/ParamPn*1000.0, -1000 ), 1000))		 	; 
			AX_Cmd[1][14]  := REAL_TO_WORD(MIN(MAX(-ParamQfU_Qmin*ParamNbPowerCol/ParamPn*1000.0, -1000 ), 1000))		  		; 
		ELSE
			AX_Cmd[1][11]  := 0 ; 
			AX_Cmd[1][12]  := 0 ; 
			AX_Cmd[1][13]  := 0 ; 
			AX_Cmd[1][14]  := 0 ; 
		END_IF

		
		
		AX_Cmd[1][15] := REAL_TO_WORD(A1_PP.ParamNominalVoltage)	; 
		AX_Cmd[1][16] := REAL_TO_WORD(A1_SUBMV.MesDataExd.MesData.MesU)	;	
		
	// Param frequency regulation 
		AX_Cmd[1][21] := REAL_TO_WORD(ParampfF_fDbHigh*100.0)		;
		AX_Cmd[1][22] := REAL_TO_WORD(ParamPfF_Fmax*100.0)		;
		AX_Cmd[1][23] := REAL_TO_WORD(ParamPfF_FDbLow*100.0)		;
		AX_Cmd[1][24] := REAL_TO_WORD(ParamPfF_Fmin*100.0)		;
		AX_Cmd[1][25] := REAL_TO_WORD(ParampfF_fDbHigh*100.0)		;
		AX_Cmd[1][26] := REAL_TO_WORD(ParamPfF_FDbLow*100.0)		;
		
		AX_Cmd[1][27] := REAL_TO_WORD(ParamPfF_FhystLow*100.0)	;
		AX_Cmd[1][28] := REAL_TO_WORD(ParamPfF_FhystHigh*100.0)	;		
		
		AX_Cmd[1][29] := REAL_TO_WORD(MIN(MAX(ParamPfF_PDbHigh/ParamPn*1000.0 , -1000 ), 1000)	)	;
		AX_Cmd[1][30] := REAL_TO_WORD(MIN(MAX(ParamPfF_Pmin/ParamPn	*1000.0, -1000 ), 1000)	)		;  
		AX_Cmd[1][31] := REAL_TO_WORD(MIN(MAX(ParamPfF_PDbLow/ParamPn*1000.0, -1000 ), 1000)	)		; 
		AX_Cmd[1][32] := REAL_TO_WORD(MIN(MAX(ParamPfF_Pmax/ParamPn*1000.0, -1000 ), 1000)		)	;  
		AX_Cmd[1][33] := REAL_TO_WORD(MIN(MAX(ParamPfF_PDbHigh/ParamPn*1000.0, -1000 ), 1000)	)		;		// P5 . 
		AX_Cmd[1][34] := REAL_TO_WORD(MIN(MAX(ParamPfF_PDbLow/ParamPn*1000.0, -1000 ), 1000)	)		; 


		AX_Cmd[1][35] := TIME_TO_WORD(ParamTimeSoCRangeReachedRmp/1000*10);				// (s) Time to go to 0 power (if SoC issue or if end of stable)
		AX_Cmd[1][37] := TIME_TO_WORD(ParamTimeEnterStblPriorRmp/1000*10);					// (s) Time to wait after entering the stable before ramping the P back to the setpoint
		AX_Cmd[1][36] := TIME_TO_WORD(ParamTimeFreqRegStbDuration/1000*10);				// (s) Time to stay in the stable area before it goes to 0
		
	// Function Mode
		AX_Cmd[1][38].0:= IN_CmdWatchdog; 							// PCS stops (hard stop) if watchdog does not change during more than 10sec
		AX_Cmd[1][38].1:= TP_Reset.Q;							// Reset
		AX_Cmd[1][38].2:= MesDataExd.OUT_CmdGridMode;	 				// To be tested
		AX_Cmd[1][38].3:= ParamSetPtModbusMode;					// Write 1 to send Setpoint via Modbus 
		AX_Cmd[1][38].4:= MesDataExd.OUT_CmdGridMode;				// Write 1 to switch to Master (to be tested)
		AX_Cmd[1][38].5:= MesDataExd.MesData.OUT_CmdStart; 				// Start: pas besoin de maintenir
		AX_Cmd[1][38].6:= MesDataExd.MesData.OUT_CmdStop; 					// Hard Stop : Open everything and stop charger .
		AX_Cmd[1][38].7:= MesDataExd.OUT_CmdP;						// P regulation enabled 
		AX_Cmd[1][38].8:= MesDataExd.OUT_CmdFreqregMode; 			// Send one to activate the Frequency regulation, to be tested
		AX_Cmd[1][38].9:= MesDataExd.OUT_CmdUregMode; 				// Send one to activate the voltage regulation, to be tested
		AX_Cmd[1][38].10:= MesDataExd.OUT_CmdQ;	 				// Q regulation enabled 
		AX_Cmd[1][38].11:= MesDataExd.OUT_CmdCosPhi;				// Cmd CosPhi ack
		AX_Cmd[1][38].12:= NOT ParamPoverQ;						// Param Q over P for Jema
		AX_Cmd[1][38].13:= ParamLVRT_Enabled;					// Param LVRT enable
		AX_Cmd[1][38].14:= ParamAntiIslanding_Enabled;			// Param Anti Islanding enable
		AX_Cmd[1][38].15:= MesDataExd.MesData.OUT_CmdStandby;				// Cmd Standby
		
		
	// Param Frequency regulation (2)
		AX_Cmd[1][39] := REAL_TO_WORD(DataSystemBMS.MesData.MesUdc);
	 
		AX_Cmd[1][40] := BOOL_TO_WORD(ParamDeactivateWatchdog);
	
		AX_Cmd[1][41].0 := NOT MesDataExd.OUT_CmdGridMode;
		
	// Setpoints

		AX_Cmd[2][1] := REAL_TO_WORD(MesDataExd.MesData.OUT_SetptP);					// Setpoint active power in kW
		AX_Cmd[2][2] := REAL_TO_WORD(MesDataExd.MesData.OUT_SetptQ);					// Setpoint reactive power in kVar
		AX_Cmd[2][4] := REAL_TO_WORD(MesDataExd.OUT_SetptCosPhi*1000);			// Setpoint CosPhi
		
	
//MesBatInit := DataSystemBMS.		

		AX_Cmd[2][18] := REAL_TO_WORD(DataSystemBMS.MesData.MesSoH);
		AX_Cmd[2][19] := REAL_TO_WORD(DataSystemBMS.MesUdcMin*1000);
		AX_Cmd[2][22] := REAL_TO_WORD(DataSystemBMS.MesUdcMax*1000);
		AX_Cmd[2][25] := UINT_TO_WORD(DataSystemBMS.MesNbRackConnected);
		AX_Cmd[2][26] := UINT_TO_WORD(DataSystemBMS.MesNbRackTot);
		AX_Cmd[2][28] := REAL_TO_WORD(DataSystemBMS.MesData.MesIdc*10);

		
		AX_Cmd[3][1] := REAL_TO_WORD(MesDataExd.OUT_SetptV);
		AX_Cmd[3][2] := REAL_TO_WORD(MesDataExd.OUT_SetptF*100);
		AX_Cmd[3][3] := REAL_TO_WORD(ParamFLow_droop*100);
		AX_Cmd[3][4] := REAL_TO_WORD(ParamFHigh_droop*100);
		AX_Cmd[3][5] := REAL_TO_WORD(ParamULow_droop); 
		AX_Cmd[3][6] := REAL_TO_WORD(ParamUHigh_droop);
		
		
// WRITE COMMAND //
	FOR KK := 1 TO 3 DO
		CmdWrite[KK] := ClockWrite OR Trig_Write[KK].Q;
	END_FOR
	
	// MODBUS REQUEST //	
		// Modbus Blocks write			
		ModbusWrite[1]
		(
			nTCPport			:= ParamTcpPort,
			pSrcAddr 			:= ADR(AX_Cmd[1]) ,
			cbLength			:= SIZEOF(AX_Cmd[1]) , 
			nQuantity 			:= AX_QTY[1],			
			Reset				:= CmdClearFault_G, 
			sIPAddr				:= ParamIPAddress , 
			nUnitID				:= ParamUnitID , 
			nMBAddr				:= AX_Adr[1] , 
			tTimeout			:= ParamTimeout ,
			WriteCmd			:= (ClockWrite OR Trig_Write[2].Q) AND MesDataExd.Mesdata.MesCP_Write , 
			ModbusWriteAlarm	=> MesModbusWriteCmdAlarm[1] , 
			ErrorId				=> MesModbusWriteCode[1]
		);   
			
		// Modbus Blocks write			
		ModbusWrite[2]
		(
			nTCPport			:= ParamTcpPort,
			pSrcAddr 			:= ADR(AX_Cmd[2]) ,
			cbLength			:= SIZEOF(AX_Cmd[2]) , 
			nQuantity 			:= AX_QTY[2],			
			Reset				:= CmdClearFault_G, 
			sIPAddr				:= ParamIPAddress , 
			nUnitID				:= ParamUnitID , 
			nMBAddr				:= AX_Adr[2] , 
			tTimeout			:= ParamTimeout ,
			WriteCmd			:= (ClockWrite OR Trig_Write[2].Q)  AND MesDataExd.Mesdata.MesCP_Write , 
			ModbusWriteAlarm	=> MesModbusWriteCmdAlarm[2] , 
			ErrorId				=> MesModbusWriteCode[2]
		);   				
		
		ModbusWrite[3]
		(
			nTCPport			:= ParamTcpPort,
			pSrcAddr 			:= ADR(AX_Cmd[3]) ,
			cbLength			:= SIZEOF(AX_Cmd[3]) , 
			nQuantity 			:= AX_QTY[3],			
			Reset				:= CmdClearFault_G, 
			sIPAddr				:= ParamIPAddress , 
			nUnitID				:= ParamUnitID, 
			nMBAddr				:= AX_Adr[3] , 
			tTimeout			:= ParamTimeout ,
			WriteCmd			:= (ClockWrite OR Trig_Write[3].Q)  AND MesDataExd.Mesdata.MesCP_Write , 
			ModbusWriteAlarm	=> MesModbusWriteCmdAlarm[3] , 
			ErrorId				=> MesModbusWriteCode[3]
		); 		
		
		
// ANALOG CMD 
OUT_SetptP_IO		:= REAL_TO_INT((32767-0)/(2*ParamPn)* MesDataExd.MesData.OUT_SetptP+32767/2) ;
OUT_SetptQ_IO		:= REAL_TO_INT((32767-0)/(2*ParamPn)* MesDataExd.MesData.OUT_SetptQ+32767/2) ;
END_METHOD

END_FUNCTION_BLOCK

// ---- 01_Equipement_Library/PCS/FB_PCS_PE.TcPOU
FUNCTION_BLOCK FB_PCS_PE EXTENDS FB_PCS_Base
//////////////////
// PLC controller . Jema Object 
//////////////////

VAR_INPUT PERSISTENT
	// Parameters of the Object
		ParamPrange							: REAL := 1559.0 ; (* (kW) Power range for scaling . *)

		ParamPn							: REAL := 1500.0;	(* (kW) Nominal power*)
		ParamPPcs						: REAL := 1265.0;
		ParamP							: REAL := 800;
		ParamQn							: REAL := 1500.0;	(* (kW) Nominal power*)
		ParamSmax							: REAL := 1500.0;	(* (kVA) Maximum apparent power of the PCS (lasts 30s)*)
		                       		
		ParamPoverQ							: BOOL := TRUE;		(* If P over Q is True, then Max setpoint for Q calculated from setpoint of P*)
    	                    			

		
 		ParamTempoStandby				: TIME	:= T#10S;	(* (s) Tempo to let time for PCS to apply a 0 setpoint before stopping . *)

     	         	    		
		ParamTimeSoCRangeReachedRmp			: TIME;				(* (ms) Time to ramp P back to the setpoint after the SoC reached its limits*)
		ParamTimeFreqRegStbDuration			: TIME;				(* (ms) Time to wait after entering the stable before ramping the P back to the setpoint *)
		ParamTimeStblRmp					: TIME; 			(* (ms) Time to ramp P back to the setpoint after entering the stable *)
		    
    {attribute 'OPC.UA.DA' := '1'}                		
		ParamAllowRechargeLowSoc			: BOOL := TRUE;		(* (NA) if true, the PCS will charge when SoC between Soc_Min and Soc_Stop*)
    {attribute 'OPC.UA.DA' := '1'}                		
		ParamPrechargeLowSoc				: REAL := 30;		(* (kW) setpoint sent at low SoC*)
    {attribute 'OPC.UA.DA' := '1'}                		
		ParamTimeLowSocToRecharge			: TIME := T#5M;		(* (ms) Time elapsed in low soc area before a soft stop is sent again *)

		ParamDeactivateWatchdog				: BOOL := TRUE;				(* Parameter to deactivate the watchdog*)

    {attribute 'OPC.UA.DA' := '1'}                		
		ParamSocLow							: REAL := 10;		(* (%) SoC from which we start limiting the maximal output Power*)
    {attribute 'OPC.UA.DA' := '1'}                		
		ParamSocHigh						: REAL := 85;		(* (%) SoC from which we start limiting the minimal output Power*)
    {attribute 'OPC.UA.DA' := '1'}                		
		ParamSocMin_G						: REAL := 5;		(* (%) Minimal SoC *)	
    {attribute 'OPC.UA.DA' := '1'}                		
		ParamSocMax_G						: REAL := 90;		(* (%) Maximal SoC *)	
    {attribute 'OPC.UA.DA' := '1'}                		
		ParamVdcStop						: REAL := 2.65;		(* (V) Vdcmin from which we stop the PCS*)
    {attribute 'OPC.UA.DA' := '1'}                		
		ParamVdcRecharge					: REAL := 2.68;		(* (V) Vdcmin from which we force the recharge*)
    {attribute 'OPC.UA.DA' := '1'}
		ParamVdcRechargeOK					: REAL := 2.7;		(* (V) Vdcmin from which we force the recharge*)
    {attribute 'OPC.UA.DA' := '1'}
		ParamVdcMin							: REAL := 1100;		(* (V) Vdcmin when we stop the forced recharge*)
    {attribute 'OPC.UA.DA' := '1'}
		ParamVdcLow							: REAL := 1150;		(* (V) VdcLow*)
    {attribute 'OPC.UA.DA' := '1'}
		ParamVdcMax							: REAL := 1300;		(* (V) VdcMax *)
    {attribute 'OPC.UA.DA' := '1'}
		ParamVdcHigh						: REAL := 1280;		(* (V) VdcHigh*)
    {attribute 'OPC.UA.DA' := '1'}
		ParamSocRecharge					: REAL := 4;		(* (%) SoC from which we recharge the PCS*)	
    {attribute 'OPC.UA.DA' := '1'}                		
		ParamSocRecharged					: REAL :=ParamSocMin_G+0.02*ParamSocMin_G;	(*(%) Soc from which we stop recharging the PCS*)
	{attribute 'OPC.UA.DA' := '1'}
		ParamPCharge						: REAL := -10;		(* (kW) power at which we consider the PCS Recharges*)
	{attribute 'OPC.UA.DA' := '1'}
		ParamChargeEfficiency				: REAL := 97;		(* (%) percentage of efficiency of PCS during charge*)
    {attribute 'OPC.UA.DA' := '1'}                		
		ParamDischargeEfficiency			: REAL := 97;		(* (%) percentage of efficiency of PCS during discharge*)
		
		ParamNbDU							: BYTE:=10 ; 			(* (NA) Total Number of disconnecting units (cables wired on the PCS)				*)
		ParamNbDU_PowerCol					: ARRAY[1..3] OF BYTE := [5,5,5]; (* (NA ) Number of disconnecting uits for each Power Columns *)
 		ParamSetpt_PCS_Discharge			:REAL;				(*SetptP parameter for the PCS discharge, if not given, it is equal to Pnom/4*)
		ParamSetpt_PCS_Charge				:REAL;  			(*SetptP parameter for the PCS charge, it is equol to 0.2*Pnom*)
		CP_PCSStop							:BOOL;
		CP_PCSStart							:BOOL;
		ParamSocStop						:REAL;
	     			
END_VAR 
VAR_INPUT   	                   			
	// Commands :

		IN_CmdPcsInLocalMode				: BOOL;				// PCS is not included in available PCS' pool (excluded from HPP control). 
		IN_CmdStopOperation					: BOOL;				// BESS Specific command : Stop operation		
		IN_CmdPreventStart					: BOOL;				// BESS Specific command : Prevent start	



		
		IN_CmdWatchdog						: BOOL ; 			// Activate or Deactivate the Watchdog function
	         
		IN_SetptCCLBat1						: REAL ; // (A) Maximal Charging Current For DC Input 1 
		IN_SetptCCLBat2						: REAL ; // (A) Maximal Charging Current For DC Input 2 
		IN_SetptCCLBat3						: REAL ; // (A) Maximal Charging Current For DC Input 3      
		IN_SetptDCLBat1						: REAL ; // (A) Maximal Discharging Current For DC Input 1 
		IN_SetptDCLBat2						: REAL ; // (A) Maximal Discharging Current For DC Input 2 
		IN_SetptDCLBat3						: REAL ; // (A) Maximal Discharging Current For DC Input 3      
		
		IN_CmdDisableCharge					: BOOL ; // Disable Charge ( SoC High reached )
		IN_CmdDisableDischarge				: BOOL ; // Disable Discharge ( SoC Low reached )
		IN_CmdLocalSocCalibration				: BOOL ; (*Launch Soc Calibration locally without needing the EMS*)
		IN_CmdEmsSocCalibration				: BOOL ; (*Launch Soc Calibration after EMS' orders*)
		IN_CmdTransfoSurcharge				: BOOL ;
		 
		IN_BMS_Selected						: WORD := 3;
		ParamDiff							:REAL;  	
		MesDataExd								: PCS_PE ;	
END_VAR
VAR_OUTPUT
	//Child objects
		OUT_SetptP_IO					: INT;			// (NA) Analogical value for the active power setpoint (based on ParamPnom)
		OUT_SetptQ_IO					: INT;			// (NA) Analogical value for the reactive power setpoint (based on ParamQnom)
END_VAR
VAR          



                           	
	//M_ALARMMANAGEMENT VARIABLES//  
		AX_AlarmWords						: ARRAY[1..30] OF ST_ValuesAlarms;
		AX_AlarmWords_Null					: ARRAY[1..30] OF ST_ValuesAlarms;
		AX_AlarmWordsJema					: ARRAY[1..225] OF ST_ValuesAlarms;
		AX_AlarmWordsJema_Null				: ARRAY[1..225] OF ST_ValuesAlarms;
		NumAlarmsActive						: UINT;
		NumAlarmsActiveJema					: UINT;
	//M_READ VARIABLES//            		
		FB_ModbusRead	          	: ARRAY[1..8] OF FB_ModbusRead; // (NA) FB for Modbus Reading
		AX_ModbusReadAlarm			: ARRAY[1..8] OF BOOL;
		AX_ModbusReadAlarmId		: ARRAY[1..8] OF UDINT;	
		
		FB_ModbusRead_PowerCol		: ARRAY[1.. CstNbPowerCol_PCS_G] OF FB_ModbusRead; 
		AX_ModbusReadAlarmPowerCol	: ARRAY[1.. CstNbPowerCol_PCS_G] OF BOOL;
		AX_ModbusReadAlarmIdPowerCol: ARRAY[1.. CstNbPowerCol_PCS_G] OF UDINT ;
		
		FB_ModbusWrite				: ARRAY[1..10]  OF FB_ModbusWrite;
		AX_ModbusWriteAlarm			: ARRAY[1..10]  OF BOOL;
		AX_ModbusWriteAlarmId		: ARRAY[1..10]  OF UDINT;	

		FB_ModbusRead_DU			: ARRAY[1..CstNbDU_PCS] OF FB_ModbusRead;
		AX_ModbusReadAlarmDU		: ARRAY[1.. CstNbDU_PCS] OF BOOL;
		AX_ModbusReadAlarmIDU		: ARRAY[1.. CstNbDU_PCS] OF UDINT ;	
	
		MesBlock_Temp_1 			: ARRAY [1..120] OF WORD ; 		// (NA) Temporary Block with multiple modbus reading 
		MesBlock_Temp_2 			: ARRAY [1..120] OF WORD ; 		// (NA) Temporary Block with multiple modbus reading 
		MesBlock_Temp_3 			: ARRAY [1..120] OF WORD ; 		// (NA) Temporary Block with multiple modbus reading 
		MesBlock_Temp_4 			: ARRAY [1..120] OF WORD ; 		// (NA) Temporary Block with multiple modbus reading 
		MesBlock_Temp_5 			: ARRAY[1..6] OF ARRAY [1..120] OF WORD ; 		// (NA) Temporary Block with multiple modbus reading 
		MesBlock_Temp_6 			: ARRAY[1..CstNbDU_PCS] OF ARRAY [1..6] OF WORD ; 		// (NA) Temporary Block with multiple modbus reading 
		MesBlock_Temp_7				: ARRAY [1..120] OF WORD ; 		// (NA) Temporary Block with multiple modbus reading 
		MesBlock_Temp_8				: ARRAY [0..120] OF BOOL ;

		
		MesBlockWrite1_Temp 			: WORD;							// (NA) Temporary Block with multiple modbus writing (Caution : Double Word variables)
		MesBlockWrite1_Temp_Old 		: WORD;							// (NA) Temporary Block with multiple modbus writing (Caution : Double Word variables)
		MesBlockWrite2_Temp				: ARRAY[1..3]    OF WORD;		// (NA) Temporary Block with multiple modbus writing (Caution : Double Word variables)
		MesBlockWrite2_Temp_Old			: ARRAY[1..3]    OF WORD;		// (NA) Temporary Block with multiple modbus writing (Caution : Double Word variables)
		MesBlockWrite3_Temp				: WORD;							// (NA) Temporary Block with multiple modbus writing (Caution : Double Word variables)
		MesBlockWrite3_Temp_Old			: WORD;							// (NA) Temporary Block with multiple modbus writing (Caution : Double Word variables)
		MesBlockWrite4_Temp				: WORD;		// (NA) Temporary Block with multiple modbus writing (Caution : Double Word variables)
		MesBlockWrite4_Temp_Old			: WORD;		// (NA) Temporary Block with multiple modbus writing (Caution : Double Word variables)
		MesBlockWrite5_Temp				: ARRAY[1..2]   OF WORD;		// (NA) Temporary Block with multiple modbus writing (Caution : Double Word variables)
		MesBlockWrite5_Temp_Old			: ARRAY[1..2]   OF WORD;		// (NA) Temporary Block with multiple modbus writing (Caution : Double Word variables)
		MesBlockWrite6_Temp				: ARRAY[1..6]   OF WORD;		// (NA) Temporary Block with multiple modbus writing (Caution : Double Word variables)
		MesBlockWrite6_Temp_Old			: ARRAY[1..6]   OF WORD;		// (NA) Temporary Block with multiple modbus writing (Caution : Double Word variables)
		MesBlockWrite7_Temp				: ARRAY[1..1]   OF WORD;		// (NA) Temporary Block with multiple modbus writing (Caution : Double Word variables)
		MesBlockWrite7_Temp_Old			: ARRAY[1..1]   OF WORD;		// (NA) Temporary Block with multiple modbus writing (Caution : Double Word variables)
		MesBlockWrite8_Temp				: BOOL ;
		MesBlockWrite9_Temp				: WORD;
		MesBlockWrite10_Temp			: WORD;
		TRIG_Write						: ARRAY[1..3] OF R_TRIG;

		AX_PcsHeartbit					: ARRAY [1..4] OF BOOL;
		                                
		TON_AlarmPcs					: ARRAY [1..CstNbPowerCol_PCS_G] OF TON ; 			// DesInhibate undervoltage alarms on PCS few seconds after PCS connected .  
                                    	                          	                                     
	                                    
		FB_SplitWordToByte				: FB_SplitWordToByte ; 			
                                        
	// M_EVALUATE VARIABLES//           
		MesStatusWatchdog					: BOOL;
		MesHeartbeat_Old					: WORD;
		Trig_Watchdog						: R_TRIG;
		Time_Discharge_LowSoc				: TIME;
		Time_Start_Discharge_LowSoc			: TIME;
		DataSystemBMS1						: BAT_SAFT;
		DataSystemBMS2						: BAT_SAFT;
		
	// Microcycling //
		MesMicroCyclingP					: REAL;				// (kW) Actual P for microcyling mode (if micro act = either ParamPmicro/-ParamPmicor, else 0)		
		MesMicroCyclingP_Old				: REAL;				// (kW) Active power the PCS will have during microcyling
	    MesMicroCyclingAllowed				: BOOL;				// (NA) If SoC is in range for microCycling                        		
		Trig_MicroCyclingNoLongerAllowed	: F_TRIG;			// Trig to detect falling edge of microcylingAllowed

	//M_WRITECOMMAND VARIABLES//    		
		TRIG_CmdOpenAC						: R_TRIG;										// Trig to detect an order to change Mode
		TRIG_CmdOpenDC						: R_TRIG;										// Trig to detect an order to change Mode
		TRIG_CmdReset						: R_TRIG;		

		TRIG_CmdStop						: R_TRIG;
		TRIG_CmdStandby						: R_TRIG;
		TRIG_CmdStart						: R_TRIG;
		TRIG_CmdPcsLocal					: R_TRIG;
		TRIG_LowLowSoC						: R_TRIG;
		TRIG_WriteToChangeModule			: R_TRIG;
		TRIG_ReadModule						: F_TRIG;
		CTU_ModuleNumber					: CTU;		
                            		
		TP_CmdBlackStart					: TP;				// TP To ensure R trig is detected
		TP_Reset							: TP ; 				// (NA) Maintain Reset command for a certain time 
		TP_CmdStandby						: TP;				// TP To maintain a soft stop order
		TP_Cmd_alarm						: TP;
		TP_CmdStandbyNow					: TP;
		TP_CmdStandbyRackEND				: TP;
		TP_Start							: TP;
		TRIG_StandbyNow						: R_TRIG;
		TRIG_StandbyRack					: R_TRIG;
		TRIG_StandbyRackEND					: R_TRIG;
		F_TRIG_StandbyRack					: F_TRIG;
		F_TRIG_END							: F_TRIG;
		F_TRIG_StandbyRackEND				: F_TRIG;
		TP_CmdStandbyRack					: TP;
		TRIG_Recharge_LowSoc				: R_TRIG;
		TRIG_RechargeBackToNormalSoc		: R_TRIG;
		TRIG_SocStop						: R_TRIG;
		TON_SocStop							: TON;
		TRIG_SocStop_Again					: R_TRIG;
        TRIG_BackToNormalSoc				: R_TRIG;
		CmdStopOperation					: BOOL;
		CmdInAlarmBat						: BOOL;
		MesAlarmsBackToNormal				: BOOL;
		xTest								: BOOL;
		F_TRIG_AlarmBat						: F_TRIG;
		// Pour la commande start, j'envoie une consigne pour fermer les contacteurs DC des batteries
		TP_CmdOpenAC						: TP;				// TP To ensure R trig is detected
		TP_CmdOpenDC						: TP;				// TP To ensure R trig is detected

		TP_CmdStart							: TP;				// TP To ensure R trig is detected
		TP_CmdPreStart						: TP;				// TP To send a close dc breaker order before sending start order
		F_TrigPreStart						: F_TRIG;			// failing edge to detect end of TP;
		
		// Pour la commande stop, pour éviter qu'on ouvre tout d'un coup, je faire un pré stop pendant 1,5s où j'envoie un autre de standby
		TP_CmdStop							: TP;				// TP To ensure R trig is detected
		TP_CmdPreStop						: TP;				// TP to send a soft stop before sending a stop 
		F_TrigPreStop						: F_TRIG;			// failing edge to detect end of TP;
		                            	

		TON_CmdStart			    		: TON;
		TON_CmdStop	                		: TON;
		TON_CmdStandby		        		: TON;

		Trig_Local_Start				: R_Trig;
		Trig_Local_Stop					: R_Trig;
		Trig_Local_EmergencyStop		: R_Trig;
		Trig_Start						: R_Trig;
		Trig_Stop						: R_Trig;
		Trig_Reset						: R_Trig;		


		F_TRIG_Standby: F_TRIG;
		F_TRIG_alarm:F_TRIG;
		F_TRIG_SoftStop:F_TRIG;		                            		

		
	
		TP_CmdStandbyDelay					: TP ; 				// TP to delay application of standby order
		
		
		
		bMaintainStop					: BOOL;	// Allow to keep setpoint to zero after a standby order .   RS .     	

		FB_Ramp_Standby			: FB_Ramp;	// Ramp to zero after a standby order
		FB_Ramp_StandbyQ		: FB_Ramp; // Ramp to zero after a standby order
	
			
		
		RS_hystlimitmin1					: RS;
		RS_hystlimitmax1					: RS;
		RS_hystlimitmin2					: RS;
		RS_hystlimitmax2					: RS;
 		RS_hystlimitEnergyShifmin			: RS;
		RS_hystlimitEnergyShifmax			: RS;
		
		CalPmaxCorr_highSoC1				: REAL;
		CalPminCorr_lowSoC1					: REAL;
		CalPmaxCorr_highSoC2				: REAL;
		CalPminCorr_lowSoC2					: REAL;
        	
		MesRead_Module_Number				: UINT;
		StartStop_RTrig				: R_Trig;
        // M_Calibration//
		CP_Calibration_Discharge		:BOOL; 			(*Boolean that has the condition  until when we should discharge*)
		CP_Calibration_Charge			:BOOL; 			(*Boolean that has the condition  until when we should consider the PCS charged*)
		FTrig_Discharge					: F_TRIG;		(*The Ftrig discharge will detect the descendent front and gives the Q = TRUE*)
		TP_Discharge					: TP;			(*The TP is used once the signal is TRUE, the TP's output stays true for 20minutes*)
		TP_Discharge_End				: TP;			(*The TP is used to detect the end of 20 minitus and thus change to the state to go to the recharge phase*)
		TON_Timeout_Calibration			: TP;			(*Time Out if the calibration takes too much time*)
		Trig_Timeout_Calibration		: F_TRIG;		(*Triggers the time out of calibration*)
		
		//SURCHARGE Transfo 
		TP_Surcharge 						: TP;	(*Timer to count 3 hours starting S of the PCS > S of the transformer allower*)				
		FTrig_Surcharge 					: F_TRIG;	(*Descendant front to detect the end of the 3 hours*)
		TransfoDurationSurchargeEnd			: BOOL;		(* (Nan) TRUE : it's been three hours that the transfo is surcharged FALSE otherwise*)
		MesTransfoSurchargeState			: BOOL;		(* (Nan) TRUE : The transfo is surcharged, False otherwise*)
		ParamSmaxTransfo					: INT :=1600;		(*The maximum apparent power accepted by the transformer*)   

		//Rack fault//
		MesStateFaultRack					: BOOL ;                            		
END_VAR

METHOD M_AlarmManagement
//////////////////
//  PCS Alarm Management 
/////////////////

VAR 
	// Method local variables (reinitialized at each cycle) 
	FB_AlarmCodeManager : FB_AlarmCodeManager ; 
	KK					: UINT;				// For Loop
	ComWarning			: BOOL;				// Aggregated Wcommunication warning
	ComAlarm			: BOOL;				// Aggregated communication Alarm
	
	CalAlarmPcsSynthesis: BOOL;
	LL					: UINT;
	ID_Journal			: UINT;
	WordTest			: WORD;
	MesNbMots			: UINT;
END_VAR
// COMMUNICATION //
	ComWarning 				:=  AX_ModbusReadAlarm[1] OR AX_ModbusReadAlarm[2] OR AX_ModbusReadAlarm[3] OR AX_ModbusReadAlarm[4] OR AX_ModbusReadAlarm[5] OR AX_ModbusReadAlarm[6] OR AX_ModbusReadAlarm[7];		
	ComAlarm				:=  AX_ModbusReadAlarm[1] AND AX_ModbusReadAlarm[2] AND AX_ModbusReadAlarm[3] AND AX_ModbusReadAlarm[4] AND AX_ModbusReadAlarm[5] AND AX_ModbusReadAlarm[6] AND AX_ModbusReadAlarm[7] ;

	FOR KK := 1 TO CstNbPowerCol_PCS_G DO
		ComWarning 	:= ComWarning OR AX_ModbusReadAlarmPowerCol[KK];
		ComAlarm	:= ComAlarm AND AX_ModbusReadAlarmPowerCol[KK];		
	END_FOR

	
		
	TON_ComAlarm(IN:= ComAlarm , PT:= ParamTempoComAlarm, Q=>MesComAlarm) ;	
	TON_ComWarning(IN := ComWarning, PT := ParamTempoComWarning, Q => MesComWarning);

	MesDataExd.MesData.MesAlarmCom		:= MesComAlarm ; 
	MesDataExd.MesData.MesWarningCom 	:= MesComWarning ; 

// PCS ALARM INHIBITION
FOR KK := 1 TO ParamNbPowerCol DO
	TON_AlarmPcs[KK](IN:=NOT MesDataExd.MesData.MesState.0, PT:= T#5S ) ;
END_FOR	


// SYNTHESES ALARMES //
CalAlarmPcsSynthesis := FALSE ; 
FOR KK:= 1 TO ParamNbPowerCol DO  
	CalAlarmPcsSynthesis := CalAlarmPcsSynthesis OR MesDataExd.AX_PowerCol[KK].MesIDState >16 ; 
END_FOR

// AlarmCode

// Attention une alarm doit être mise en commentaire de la manière suivante (* *), l'utilisation du // pose pb sur Bazefield 	
	
	FB_AlarmCodeManager(
		bAlarm1		:= CalAlarmPcsSynthesis		,								// Power columns Alarm Synthesis, at least one alarm active on power column
		bAlarm2		:= FALSE , //
		bAlarm3		:= FALSE , //	
		bAlarm4		:= FALSE,										            //                              			    	
		bAlarm5		:= FALSE , //
		bAlarm6		:= FALSE , //                 				
		bAlarm7		:= FALSE , //
		bAlarm8 	:= FALSE , //
		bAlarm9		:= FALSE , //
		bAlarm10	:= FALSE , //
		bAlarm11	:= MesDataExd.MesData.MesAlarmCom,                                     // Communication alarm : none of the Power Columns are responding 				
		bAlarm12	:= MesDataExd.MesData.MesAlarm,                                               	//PCS Controller general Alarm		
		bAlarm13	:= FALSE,                                               	//			
		bAlarm14	:= FALSE,                                               	//		
		bAlarm15	:= FALSE,                                               	//		
		wAlarmCode	=>MesDataExd.MesData.MesAlarmCode);		                                		
		                                                                                 	
		
		
// WARNING CODE //
	FB_AlarmCodeManager(
		bAlarm1		:= MesComWarning, 																											// Communication warning : At least one of the Power Columns are not responding 
		bAlarm2		:= MesDataExd.MesData.MesWarning,																							//PCS Controller general Warning  
		bAlarm3		:= MesDataExd.MesIDState = 10  ,  																							// LVRT is running 
		bAlarm4		:= MesDataExd.MesIDState = 11,    																							// OVRT is runnning
		bAlarm5		:= FALSE , // 
		bAlarm6		:= FALSE , // 
		bAlarm7		:= FALSE , // 
		bAlarm8		:= FALSE , // 
		bAlarm9		:= FALSE , // 
		bAlarm10	:= FALSE , // 
		bAlarm11	:= FALSE , // 
		bAlarm12	:= FALSE , // 
		bAlarm13	:= FALSE,           																										//
		bAlarm14	:= FALSE,           																										//
		bAlarm15	:= FALSE,           																										//
		wAlarmCode	=>MesDataExd.MesData.MesWarningCode);
		
// EVENT CODE //
	FB_AlarmCodeManager(
		bAlarm1			:= FALSE , // 
		bAlarm2			:= MesDataExd.MesData.MesOpened_Dc, 																											// DC Switch Closed
		bAlarm3			:= MesDataExd.MesData.OUT_CmdStandby, 																												// Soft stop command
		bAlarm4			:= MesDataExd.MesData.MesOnGrid,																													// OnGrid Mode is activated
		bAlarm5			:= MesDataExd.MesData.MesOffGrid, 																													// Offgrid Mode is activated
		bAlarm6			:= MesDataExd.MesData.OUT_CmdStart, 																												// Cmd Start
		bAlarm7			:= MesDataExd.MesData.OUT_CmdStop, 																												// Full stop command
		bAlarm8			:= FALSE , // 
		bAlarm9			:= FALSE , // 
		bAlarm10		:= FALSE , // 
		bAlarm11		:= FALSE , // 
		bAlarm12		:= MesDataExd.MesData.MesOpened_Ac, 																											// Ac breaker is Closed. 
		bAlarm13		:= FALSE , //
		bAlarm14		:= FALSE , //
		bAlarm15		:= FALSE , //
		wAlarmCode		=>MesDataExd.MesData.MesEventCode);                                                                                           					// 
		

NumAlarmsActive := 0;
AX_AlarmWords := AX_AlarmWords_Null;
MesNbMots := 2;
FOR KK := 1 TO MesNbMots DO			// Combien j'ai de mots
	ID_Journal := 15 + (ParamEssNum-1) * MesNbMots * CstNbPcs_ESS_G + (ParamPcsNum - 1) * CstNbPcs_ESS_G + (KK- 1);
	FOR LL := 1 TO 15 DO 	// Les bits 
		WordTest := ROR(FUN_Alarms.AX_RecupWord[ID_Journal],LL);
		IF WordTest.0 THEN
			NumAlarmsActive := NumAlarmsActive + 1;
			AX_AlarmWords[NumAlarmsActive].Message := FUN_Alarms.AX_Journal[ID_Journal][LL].Message;
		ELSE
			AX_AlarmWords[NumAlarmsActive+1].Message := '';
		END_IF
	END_FOR
END_FOR		

NumAlarmsActiveJema := 0;
AX_AlarmWordsJema := AX_AlarmWordsJema_Null;
MesNbMots := 15;
FOR KK := 1 TO MesNbMots DO			// Combien j'ai de mots
	FOR LL := 1 TO 15 DO 	// Les bits 
		ID_Journal := 57 + (ParamEssNum-1) * MesNbMots * CstNbPcs_ESS_G + (ParamPcsNum - 1) * CstNbPcs_ESS_G + (KK- 1);
		WordTest := ROR(FUN_Alarms.AX_RecupWord[ID_Journal],LL);
		IF WordTest.0 THEN
			NumAlarmsActiveJema := NumAlarmsActiveJema + 1;
			AX_AlarmWordsJema[NumAlarmsActiveJema].Message := FUN_Alarms.AX_Journal[ID_Journal][LL].Message;
		ELSE
			AX_AlarmWordsJema[NumAlarmsActiveJema+1].Message := '';
		END_IF
	END_FOR
END_FOR
END_METHOD

METHOD M_Calibration
VAR
	KK								: INT;
END_VAR
//SOC CALIBRATION
//Process of Calibration starting, conditions found on SAFT document
MesDataExd.MesCalibrationState.0 := 1; //Calibration Started
	FOR KK:=1 TO CstNbBat_ESS_G DO
	//	CP_Calibration_Discharge := CP_Calibration_Discharge OR (AX_ESS[ParamEssNum].AX_Bat[KK].MesDataExd.MesData.MesDCL < 36 * AX_ESS[ParamEssNum].AX_Bat[KK].MesDataExd.MesNbRackConnected AND AX_ESS[ParamEssNum].AX_Bat[KK].MesDataExd.MesIDAlarm_Vendor1.12);
	END_FOR
	
	// If the condition is not met we discharge
	IF NOT(CP_Calibration_Discharge) THEN
		MesDataExd.MesData.OUT_SetptP := ParamSetpt_PCS_Discharge;
		MesDataExd.MesCalibrationState.1 := 1; //We send the setpoint to the PCS, the PCS starts discharging
	END_IF
	
	//If the condition is met we stop the discharge and change the calibration state of the pcs
	IF CP_Calibration_Discharge THEN
		MesDataExd.MesCalibrationState.2 := 1; //Discharging done and starting 20min hold
	END_IF
	//By changing the calibration state of the PCS we can start holding off the PCS for 20min
	IF MesDataExd.MesCalibrationState.2 THEN
		TP_Discharge(IN:=MesDataExd.MesCalibrationState.2,PT:=T#20M);
		MesDataExd.MesData.OUT_SetptP := 0;
	END_IF
	
	//Once the 20min is done, we can start charging
	FTrig_Discharge(CLK := TP_Discharge.Q);
	
	IF FTrig_Discharge.Q THEN
		MesDataExd.MesCalibrationState.3 := 1;
	END_IF
	IF MesDataExd.MesCalibrationState.3 THEN
		FOR KK:=1 TO CstNbBat_ESS_G DO
				CP_Calibration_Charge := CP_Calibration_Charge AND (AX_ESS[ParamEssNum].AX_Bat[KK].MesDataExd.MesData.MesSoC >= ParamSocRecharged);
		END_FOR
		IF NOT(CP_Calibration_Charge) THEN
			 //Charging had started
			MesDataExd.MesData.OUT_SetptP := ParamSetpt_PCS_Charge;
		END_IF
		IF CP_Calibration_Charge THEN
			MesDataExd.MesCalibrationState:=0;
		END_IF
	END_IF
END_METHOD

METHOD M_CP
//////////////////
//  Emulator
/////////////////

VAR 
	// Method local variables (reinitialized at each cycle) 
	
END_VAR
	CalCP_Stop 					:=  TRUE;
	CalCP_Start					:=  NOT MesDataExd.MesData.MesAlarmCode.0 AND NOT CmdClearFault_G AND MesDataExd.MesData.MesState.0 AND  (MesDataExd.MesIDState = 2 OR MesDataExd.MesIDState = 4)AND NOT TP_CmdStop.Q AND NOT IN_CmdStopOperation AND NOT IN_CmdPreventStart ;
	
	CalCP_Reset 				:=  TRUE;
	CalCP_Standby				:= NOT TP_CmdStop.Q  ; 



SUPER^.M_CP() ; 




Trig_Cmd_Read(CLK:=IN_CmdToggleRead);
Trig_Cmd_Write(CLK:=IN_CmdToggleWrite);
	
IF Trig_Cmd_Read.Q THEN
	IN_CmdToggleRead := FALSE;
	MesDataExd.MesData.MesCP_Read := NOT MesDataExd.MesData.MesCP_Read;
END_IF


IF Trig_Cmd_Write.Q THEN
	IN_CmdToggleWrite := FALSE;
	MesDataExd.MesData.MesCP_Write := NOT MesDataExd.MesData.MesCP_Write;
END_IF
END_METHOD

METHOD M_Evaluate : BOOL
VAR_INPUT
END_VAR
VAR
	KK : UINT;
	bTest: BOOL;
	MesAlarmPcs: BOOL;
	AX_Journal : ARRAY[57..57] OF ARRAY[1..15] OF ST_ValuesAlarms;
	CalCoeffSoC_Charge			: USINT;
	CalCoeffSoC_Discharge		: USINT;
	
	DataSystemBMS		: BAT_SAFT ; 
END_VAR
// External values update :
	DataSystemBMS1 				:= AX_ESS[ParamEssNum].AX_Bat[1].MesDataExd;
	DataSystemBMS2 				:= AX_ESS[ParamEssNum].AX_Bat[2].MesDataExd;


// Gestion des Start/Stop par SOC Low
	CP_PCSStop := (DataSystemBMS1.MesData.MesUdcMin_Cell <= ParamVdcStop) OR (DataSystemBMS2.MesData.MesUdcMin_Cell <= ParamVdcStop);
	TRIG_SocStop(clk := NOT MesDataExd.MesData.MesState.0 AND NOT MesDataExd.MesData.MesState.14 AND CP_PCSStop);
	IF TRIG_SocStop.Q THEN 
		MesDataExd.MesData.MesState.14 := TRUE;
	END_IF
	
	
	TRIG_SocStop_Again(CLK := Time_Discharge_LowSoc > ParamTimeLowSocToRecharge);
	IF NOT MesDataExd.MesData.MesState.0 AND MesDataExd.MesData.MesState.14 AND MesDataExd.MesData.MesPdc >= 0 THEN
		Time_Discharge_LowSoc := Time_Discharge_LowSoc + TIME() - Time_Start_Discharge_LowSoc;
	ELSIF MesDataExd.MesData.MesState.0 AND (NOT MesDataExd.MesData.MesState.14 OR Time_Discharge_LowSoc >= ParamTimeLowSocToRecharge) THEN
		Time_Discharge_LowSoc := T#0S;
	END_IF
	Time_Start_Discharge_LowSoc := TIME();
	CP_PCSStart := (DataSystemBMS1.MesData.MesUdcMin_Cell > ParamVdcStop) OR (DataSystemBMS2.MesData.MesUdcMin_Cell > ParamVdcStop);
	TRIG_BackToNormalSoc(CLK := MesDataExd.MesData.MesState.14 AND CP_PCSStart);
	IF TRIG_BackToNormalSoc.Q THEN
		MesDataExd.MesData.MesState.14 := 0;
	END_IF
	
	
	
	IF ParamAllowRechargeLowSoc THEN
		TRIG_Recharge_LowSoc(CLK := NOT MesDataExd.MesData.MesState.0 AND NOT MesDataExd.MesData.MesState.14 AND (DataSystemBMS1.MesData.MesUdcMin_Cell <= ParamVdcRecharge OR DataSystemBMS2.MesData.MesUdcMin_Cell <= ParamVdcRecharge));
		IF TRIG_Recharge_LowSoc.Q THEN
			MesDataExd.MesData.MesState.13 := TRUE;
		END_IF
		
		TRIG_RechargeBackToNormalSoc(CLK := MesDataexd.MesData.MesState.13 AND (DataSystemBMS1.MesData.MesUdcMin_Cell >= ParamVdcRechargeOK AND DataSystemBMS2.MesData.MesUdcMin_Cell >= ParamVdcRechargeOK));
		IF TRIG_RechargeBackToNormalSoc.Q THEN
			MesDataexd.MesData.MesState.13 := FALSE;
		END_IF
	END_IF
	
	
	
// PROPERTIES UPDATE // 



//--------------------------------------------------------------------------------//
// 							Gestion des setpoints								  //
//--------------------------------------------------------------------------------//

// Gestion des limites hautes de SoC
	RS_hystlimitmax1(SET:= DataSystemBMS1.MesData.MesUdc >= ParamVdcMax , RESET1:= DataSystemBMS1.MesData.MesUdc < ParamVdcHigh) ; 
	RS_hystlimitmin1(SET:= DataSystemBMS1.MesData.MesUdc <= ParamVdcMin , RESET1:= DataSystemBMS1.MesData.MesUdc > ParamVdcLow) ; 
	RS_hystlimitmax2(SET:= DataSystemBMS2.MesData.MesUdc >= ParamVdcMax , RESET1:= DataSystemBMS2.MesData.MesUdc < ParamVdcHigh) ; 
	RS_hystlimitmin2(SET:= DataSystemBMS2.MesData.MesUdc <= ParamVdcMin , RESET1:= DataSystemBMS2.MesData.MesUdc > ParamVdcLow) ;
	
	IF DataSystemBMS1.MesData.MesUdc >= ParamVdcHigh THEN
		CalPmaxCorr_highSoC1 := (ParamVdcMax - DataSystemBMS1.MesData.MesUdc)/(ParamVdcMax - ParamVdcHigh);
	ELSE 
		CalPmaxCorr_highSoC1 := 1 ;
	END_IF
	IF DataSystemBMS2.MesData.MesUdc >= ParamVdcHigh THEN
		CalPmaxCorr_highSoC2 := (ParamVdcMax - DataSystemBMS2.MesData.MesUdc)/(ParamVdcMax - ParamVdcHigh);
	ELSE 
		CalPmaxCorr_highSoC2 := 1 ;
	END_IF
	IF DataSystemBMS1.MesData.MesUdc <= ParamVdcLow THEN
		CalPminCorr_lowSoC1 := (ParamVdcMin - DataSystemBMS1.MesData.MesUdc)/(ParamVdcMin - ParamVdcLow );
	ELSE
		CalPminCorr_lowSoC1 := 1;
	END_IF
	IF DataSystemBMS2.MesData.MesUdc <= ParamVdcLow THEN
		CalPminCorr_lowSoC2 := (ParamVdcMin - DataSystemBMS2.MesData.MesUdc)/(ParamVdcMin - ParamVdcLow );
	ELSE
		CalPminCorr_lowSoC2 := 1;
	END_IF
	
	IF IN_BMS_Selected = 3 AND ((IN_SetptCCLBat1 <> 0 OR IN_SetptDCLBat1 <> 0) AND  AX_ESS[ParamEssNum].AX_Bat[1].MesDataExd.MesData.MesUdc <> 0) (* AND ((IN_SetptCCLBat2 <> 0 OR IN_SetptDCLBat2 <> 0) AND  AX_ESS[ParamEssNum].AX_Bat[2].MesDataExd.MesData.MesUdc <> 0)*) THEN
		MesDataExd.MesData.MesSmax_ChargeFromBat 		:=  MIN(((SEL(RS_hystlimitmax1.Q1, 1, 0)*CalPmaxCorr_highSoC1*IN_SetptCCLBat1 * AX_ESS[ParamEssNum].AX_Bat[1].MesDataExd.MesData.MesUdc*(ParamChargeEfficiency/100)) +(SEL(RS_hystlimitmax2.Q1, 1, 0)*CalPmaxCorr_highSoC2*IN_SetptCCLBat2 * AX_ESS[ParamEssNum].AX_Bat[2].MesDataExd.MesData.MesUdc)*(ParamChargeEfficiency/100))/1000,	ParamPn);
		MesDataExd.MesData.MesSmax_DischargeFromBat 	:=  MIN(((SEL(RS_hystlimitmin1.Q1, 1, 0)*CalPminCorr_lowSoC1*IN_SetptDCLBat1 * AX_ESS[ParamEssNum].AX_Bat[1].MesDataExd.MesData.MesUdc*(ParamDischargeEfficiency/100)) +(SEL(RS_hystlimitmin2.Q1, 1, 0)*CalPminCorr_lowSoC2*IN_SetptDCLBat2 * AX_ESS[ParamEssNum].AX_Bat[2].MesDataExd.MesData.MesUdc)*(ParamDischargeEfficiency/100))/1000,	ParamPn);
	
	ELSIF IN_BMS_Selected = 1 AND ((IN_SetptCCLBat1 <> 0 OR IN_SetptDCLBat1 <> 0) AND  AX_ESS[ParamEssNum].AX_Bat[1].MesDataExd.MesData.MesUdc <> 0) THEN
		MesDataExd.MesData.MesSmax_ChargeFromBat 		:=  MIN(SEL(RS_hystlimitmax1.Q1, 1, 0)*CalPmaxCorr_highSoC1*IN_SetptCCLBat1 * AX_ESS[ParamEssNum].AX_Bat[1].MesDataExd.MesData.MesUdc*(ParamChargeEfficiency/100)/1000,	ParamPn);
		MesDataExd.MesData.MesSmax_DischargeFromBat 	:=  MIN(SEL(RS_hystlimitmin1.Q1, 1, 0)*CalPminCorr_lowSoC1*IN_SetptDCLBat1 * AX_ESS[ParamEssNum].AX_Bat[1].MesDataExd.MesData.MesUdc*(ParamDischargeEfficiency/100)/1000,	ParamPn);
	
	ELSIF IN_BMS_Selected = 2 AND ((IN_SetptCCLBat2 <> 0 OR IN_SetptDCLBat2 <> 0) AND  AX_ESS[ParamEssNum].AX_Bat[2].MesDataExd.MesData.MesUdc <> 0) THEN
		MesDataExd.MesData.MesSmax_ChargeFromBat 		:=  MIN(SEL(RS_hystlimitmax2.Q1, 1, 0)*CalPmaxCorr_highSoC2*IN_SetptCCLBat2 * AX_ESS[ParamEssNum].AX_Bat[2].MesDataExd.MesData.MesUdc*(ParamChargeEfficiency/100)/1000,	ParamPn);
		MesDataExd.MesData.MesSmax_DischargeFromBat 	:=  MIN(SEL(RS_hystlimitmin2.Q1, 1, 0)*CalPminCorr_lowSoC2*IN_SetptDCLBat2 * AX_ESS[ParamEssNum].AX_Bat[2].MesDataExd.MesData.MesUdc*(ParamDischargeEfficiency/100)/1000,	ParamPn);
	ELSE 
		MesDataExd.MesData.MesSmax_ChargeFromBat := 0;
		MesDataExd.MesData.MesSmax_DischargeFromBat := 0;
	END_IF
	//IF IN_SetptCCLBat1 <> IN_SetptCCLBat2 THEN
		//MesDataExd.MesData.MesSmax_ChargeFromBat:= 2*MIN((IN_SetptCCLBat1 * AX_ESS[ParamEssNum].AX_Bat[1].MesDataExd.MesData.MesUdc)/1000,(IN_SetptCCLBat2 * AX_ESS[ParamEssNum].AX_Bat[2].MesDataExd.MesData.MesUdc)/1000);
	//END_IF
	//IF IN_SetptDCLBat1 <180 OR IN_SetptDCLBat2 < 180  THEN
	//	MesDataExd.MesData.MesSmax_DischargeFromBat:=0;
	//END_IF
	
	
	IF (DataSystemBMS1.MesData.MesCCL <> 0 OR DataSystemBMS1.MesData.MesDCL <> 0) AND DataSystemBMS1.MesData.MesUdc <> 0 THEN
		MesDataExd.MesData.MesPmax1_ChargeFromBat 		:= 1- (IN_SetptCCLBat1*AX_ESS[ParamEssNum].AX_Bat[1].MesDataExd.MesData.MesUdc)/((IN_SetptCCLBat2*AX_ESS[ParamEssNum].AX_Bat[2].MesDataExd.MesData.MesUdc) + (IN_SetptCCLBat1*AX_ESS[ParamEssNum].AX_Bat[1].MesDataExd.MesData.MesUdc));
		MesDataExd.MesData.MesPmax1_DischargeFromBat 	:=  (IN_SetptDCLBat1*AX_ESS[ParamEssNum].AX_Bat[1].MesDataExd.MesData.MesUdc)/((IN_SetptDCLBat2*AX_ESS[ParamEssNum].AX_Bat[2].MesDataExd.MesData.MesUdc) + (IN_SetptDCLBat1*AX_ESS[ParamEssNum].AX_Bat[1].MesDataExd.MesData.MesUdc));
		MesDataExd.MesData.MesPmax2_ChargeFromBat 		:= 1- (IN_SetptCCLBat2*AX_ESS[ParamEssNum].AX_Bat[2].MesDataExd.MesData.MesUdc)/((IN_SetptCCLBat2*AX_ESS[ParamEssNum].AX_Bat[2].MesDataExd.MesData.MesUdc) + (IN_SetptCCLBat1*AX_ESS[ParamEssNum].AX_Bat[1].MesDataExd.MesData.MesUdc));
		MesDataExd.MesData.MesPmax2_DischargeFromBat 	:=  (IN_SetptDCLBat2*AX_ESS[ParamEssNum].AX_Bat[2].MesDataExd.MesData.MesUdc)/((IN_SetptDCLBat2*AX_ESS[ParamEssNum].AX_Bat[2].MesDataExd.MesData.MesUdc) + (IN_SetptDCLBat1*AX_ESS[ParamEssNum].AX_Bat[1].MesDataExd.MesData.MesUdc));
	ELSE
		MesDataExd.MesData.MesPmax1_ChargeFromBat := 0;
		MesDataExd.MesData.MesPmax1_DischargeFromBat := 0;
		MesDataExd.MesData.MesPmax2_ChargeFromBat := 0;
		MesDataExd.MesData.MesPmax2_DischargeFromBat := 0;
	END_IF
// Local
	// Si je suis en local, je désactive le micro cycling et je réecris le setpoint d'input	
	IF MesDataExd.MesData.OUT_CmdPcsLocal THEN
		IN_SetptP := IN_SetptP_Local;
		IN_SetptQ := IN_SetptQ_Local;
		MesDataExd.MesData.OUT_SetptPMax :=IN_SetptP_Local;
		MesDataExd.MesData.OUT_SetptPMin :=-IN_SetptP_Local;
		MesDataExd.MesData.OUT_SetptP1Max :=IN_SetptP_Local;
		MesDataExd.MesData.OUT_SetptP1Min :=-IN_SetptP_Local;
		MesDataExd.MesData.OUT_SetptP2Max :=IN_SetptP_Local;
		MesDataExd.MesData.OUT_SetptP2Min :=-IN_SetptP_Local;
	END_IF

	
IF ParamPoverQ THEN 
	// Le setpoint Max correspond à la dispo * la puissance nominale
	IF (DataSystemBMS1.MesData.MesIDState = 3 OR DataSystemBMS1.MesData.MesIDState = 5) AND (DataSystemBMS2.MesData.MesIDState = 3 OR DataSystemBMS2.MesData.MesIDState = 3) THEN
		ParamP := 800;
	ELSE 
		ParamP := 1150;
	END_IF
	
	MesDataExd.MesData.OUT_SetptSMax := 230*(DataSystemBMS1.MesData.MesNbRackConnected+DataSystemBMS2.MesData.MesNbRackConnected); //MesDataExd.MesData.MesAvailability * MesDataExd.MesData.MesSnom/100.0
	IF NOT MesDataExd.MesCalibrationState.0 THEN
		MesDataExd.MesData.OUT_SetptPMax := MIN(MesDataExd.MesData.OUT_SetptSMax,MesDataExd.MesData.MesSmax_DischargeFromBat,((MesDataExd.MesP_DischargeMax/100)*MesDataExd.MesData.OUT_SetptSMax),ParamPn);
		MesDataExd.MesData.OUT_SetptPMin := - MIN(MesDataExd.MesData.OUT_SetptSMax,MesDataExd.MesData.MesSmax_ChargeFromBat,((MesDataExd.MesP_ChargeMax/100)*MesDataExd.MesData.OUT_SetptSMax),ParamPn);
		MesDataExd.MesData.OUT_SetptP1Max := MIN((SEL(RS_hystlimitmin1.Q1, 1, 0)*CalPminCorr_lowSoC1*(ParamDischargeEfficiency/100)*IN_SetptDCLBat1*AX_ESS[ParamEssNum].AX_Bat[1].MesDataExd.MesData.MesUdc)/1000, ParamP, ((MesDataExd.MesP_DischargeMax1/100)*MesDataExd.MesData.MesSnom));
		MesDataExd.MesData.OUT_SetptP1Min :=  - MIN((SEL(RS_hystlimitmax1.Q1, 1, 0)*CalPmaxCorr_highSoC1*(ParamDischargeEfficiency/100)*IN_SetptCCLBat1*AX_ESS[ParamEssNum].AX_Bat[1].MesDataExd.MesData.MesUdc)/1000, ParamP,  ((MesDataExd.MesP_ChargeMax1/100)*MesDataExd.MesData.MesSnom));
		MesDataExd.MesData.OUT_SetptP2Max := MIN((SEL(RS_hystlimitmin2.Q1, 1, 0)*CalPminCorr_lowSoC2*(ParamDischargeEfficiency/100)*IN_SetptDCLBat2*AX_ESS[ParamEssNum].AX_Bat[2].MesDataExd.MesData.MesUdc)/1000, ParamP ,((MesDataExd.MesP_DischargeMax2/100)*MesDataExd.MesData.MesSnom));
		MesDataExd.MesData.OUT_SetptP2Min :=  - MIN((SEL(RS_hystlimitmax2.Q1, 1, 0)*CalPmaxCorr_highSoC2*(ParamDischargeEfficiency/100)*IN_SetptCCLBat2*AX_ESS[ParamEssNum].AX_Bat[2].MesDataExd.MesData.MesUdc)/1000, ParamP,((MesDataExd.MesP_ChargeMax2/100)*MesDataExd.MesData.MesSnom));
	ELSE
		MesDataExd.MesData.OUT_SetptPMax :=0;
		MesDataExd.MesData.OUT_SetptPMin :=0;
		MesDataExd.MesData.OUT_SetptP1Max :=0;
		MesDataExd.MesData.OUT_SetptP1Min :=0;
		MesDataExd.MesData.OUT_SetptP2Max :=0;
		MesDataExd.MesData.OUT_SetptP2Min :=0;
	END_IF
	
	//Test SAFT IMD/2
	MesDataExd.OUT_SetptPMax_IMDicharge1 := MIN(IN_SetptP_Local, (IN_SetptDCLBat1*AX_ESS[ParamEssNum].AX_Bat[1].MesDataExd.MesData.MesUdc)/1000);
	MesDataExd.OUT_SetptPMAX_IMDicharge2 := MIN(IN_SetptP_Local, (IN_SetptDCLBat2*AX_ESS[ParamEssNum].AX_Bat[2].MesDataExd.MesData.MesUdc)/1000);
	MesDataExd.OUT_SetptPMax_IMCharge1 := MAX(IN_SetptP_Local, (-IN_SetptCCLBat1*AX_ESS[ParamEssNum].AX_Bat[1].MesDataExd.MesData.MesUdc)/1000);
	MesDataExd.OUT_SetptPMax_IMCharge2 := MAX(IN_SetptP_Local, (-IN_SetptCCLBat2*AX_ESS[ParamEssNum].AX_Bat[2].MesDataExd.MesData.MesUdc)/1000);
	

	
		// Min
	IF ABS(MesDataExd.MesData.OUT_SetptSMax) > ABS(MesDataExd.MesData.OUT_SetptP) THEN
		MesDataExd.MesData.OUT_SetptQMax		:= MIN(ParamQn, SQRT(EXPT(MesDataExd.MesData.OUT_SetptSMax, 2) - EXPT(MesDataExd.MesData.OUT_SetptP, 2)));
	ELSE
		MesDataExd.MesData.OUT_SetptQMax := 0;
	END_IF
	IF ABS(MesDataExd.MesData.OUT_SetptSMax) > ABS(MesDataExd.MesData.OUT_SetptP) THEN
		MesDataExd.MesData.OUT_SetptQMin		:= -MIN(ParamQn,SQRT( EXPT(MesDataExd.MesData.OUT_SetptSMax, 2) - EXPT(MesDataExd.MesData.OUT_SetptP, 2)));
	ELSE 
		MesDataExd.MesData.OUT_SetptQMin := 0;
	END_IF
	
ELSE

	MesDataExd.MesData.OUT_SetptQMax := MIN( ParamQn , MIN ( SEL(MesDataExd.MesData.MesP = 0, SEL(MesDataExd.MesData.MesP>0, MesDataExd.MesData.MesSmax_ChargeFromBat, MesDataExd.MesData.MesSmax_DischargeFromBat), MIN(MesDataExd.MesData.MesSmax_ChargeFromBat, MesDataExd.MesData.MesSmax_DischargeFromBat)),ParamQn *MesDataExd.MesData.MesAvailability /100 ));
	MesDataExd.MesData.OUT_SetptQMin := - MesDataExd.MesData.OUT_SetptQMax;
	
	MesDataExd.MesData.OUT_SetptPMax		:=MIN(ParamPn ,  MIN(MesDataExd.MesData.MesAvailability * ParamPrange/100.0,  SQRT(EXPT(MesDataExd.MesData.MesSmax_DischargeFromBat,2) - EXPT(MesDataExd.MesData.OUT_SetptQ,2)))*SEL(MesDataExd.MesData.MesState.0 , 1,0 )) ;
	MesDataExd.MesData.OUT_SetptPMin		:=MAX(-ParamPn , MAX(- MesDataExd.MesData.MesAvailability *ParamPrange/100.0 , SQRT(EXPT(MesDataExd.MesData.MesSmax_ChargeFromBat,2) - EXPT(MesDataExd.MesData.OUT_SetptQ,2)))*SEL(MesDataExd.MesData.MesState.0 , 1,0 ) );
	

END_IF

// J'affecte les variables que je vais écrire


	IF ParamAllowRechargeLowSoc AND MesDataExd.MesData.MesState.13 THEN
		IN_SetptP := MIN(-20, - ABS(ParamPrechargeLowSoc));
	END_IF
	IF IN_SetptP >= 0 AND MesDataExd.MesData.OUT_SetptPMax <>0 THEN 
		MesDataExd.MesData.OUT_SetptP1		:= MIN(IN_SetptP*MesDataExd.MesData.MesPmax1_DischargeFromBat,MesDataExd.MesData.OUT_SetptP1Max);
		MesDataExd.MesData.OUT_SetptP2		:= MIN(IN_SetptP*MesDataExd.MesData.MesPmax2_DischargeFromBat,MesDataExd.MesData.OUT_SetptP2Max);
	ELSIF IN_SetptP < 0 AND MesDataExd.MesData.OUT_SetptPMin <>0 THEN
		MesDataExd.MesData.OUT_SetptP1		:= MAX(-ABS(IN_SetptP*MesDataExd.MesData.MesPmax1_ChargeFromBat),MesDataExd.MesData.OUT_SetptP1Min);
		MesDataExd.MesData.OUT_SetptP2		:= MAX(-ABS(IN_SetptP*MesDataExd.MesData.MesPmax2_ChargeFromBat),MesDataExd.MesData.OUT_SetptP2Min);
	ELSE
		MesDataExd.MesData.OUT_SetptP1:=0;
		MesDataExd.MesData.OUT_SetptP2:=0;	
	END_IF
	
	IF (MesDataExd.AX_PowerCol[1].MesStateIO.1 <> 0 OR MesDataExd.AX_PowerCol[3].MesStateIO.1 <> 0) AND (MesDataExd.AX_PowerCol[2].MesStateIO.1 = 0 AND MesDataExd.AX_PowerCol[4].MesStateIO.1 = 0)THEN
		IF IN_SetptP >=0 THEN
			MesDataExd.MesData.OUT_SetptP1		:= MIN(IN_SetptP,MesDataExd.MesData.OUT_SetptP1Max);
			MesDataExd.MesData.OUT_SetptP2 :=0;
		ELSIF IN_SetptP <0 THEN
			MesDataExd.MesData.OUT_SetptP1		:= MAX(IN_SetptP,MesDataExd.MesData.OUT_SetptP1Min);
			MesDataExd.MesData.OUT_SetptP2 :=0;
		END_IF
	ELSIF (MesDataExd.AX_PowerCol[2].MesStateIO.1 <> 0 OR MesDataExd.AX_PowerCol[4].MesStateIO.1 <> 0) AND (MesDataExd.AX_PowerCol[1].MesStateIO.1 = 0 AND MesDataExd.AX_PowerCol[3].MesStateIO.1 = 0) THEN
		IF IN_SetptP >=0 THEN
			MesDataExd.MesData.OUT_SetptP2		:= MIN(IN_SetptP,MesDataExd.MesData.OUT_SetptP2Max);
			MesDataExd.MesData.OUT_SetptP1 :=0;
		ELSIF IN_SetptP <0 THEN
			MesDataExd.MesData.OUT_SetptP2		:= MAX(IN_SetptP,MesDataExd.MesData.OUT_SetptP2Min);
			MesDataExd.MesData.OUT_SetptP1 :=0;
		END_IF
	END_IF
	//MesDataExd.MesData.OUT_SetptP		:= MIN(MAX(IN_SetptP, MesDataExd.MesData.OUT_SetptPMin), MesDataExd.MesData.OUT_SetptPMax);
	MesDataExd.MesData.OUT_SetptQ		:= -MIN(MAX(IN_SetptQ, MesDataExd.MesData.OUT_SetptQMin), MesDataExd.MesData.OUT_SetptQMax);

//Transfo Surcharge
// Surcharge transfo //
(*Here I know that we have only one PCS if we had two PCS we would a for loop*)
	MesTransfoSurchargeState := MesDataExd.MesData.MesS > ParamSmaxTransfo; //We check if the apparent power is superior to the apparent power accepted by the transfo
	TP_Surcharge(IN:=MesTransfoSurchargeState,PT:=T#3H); //if it's true we start a 3hour timer
	FTrig_Surcharge(CLK := TP_Surcharge.Q); 
	IF FTrig_Surcharge.Q THEN
		TransfoDurationSurchargeEnd := TRUE; //We detect that these three hours ended
	END_IF
	IF TransfoDurationSurchargeEnd THEN
		MesDataExd.MesData.OUT_SetptSMax := (ParamSmaxTransfo - 0.1*ParamSmaxTransfo); //When the three hours end we immadietly send a maximum S setpoint of 10% less than the maximum allowed 
	END_IF
	IF NOT(MesTransfoSurchargeState) THEN
		TransfoDurationSurchargeEnd := FALSE; //As long as the apparent power doesnt go under the ParamSmaxTransfo we continue sending setpoints 
	END_IF
END_METHOD

METHOD M_Execute
//////////////////
//  Method Calls 
/////////////////

VAR 
	// Method local variables (reinitialized at each cycle) 
	KK			: BYTE;			// For Loop 
	
END_VAR
// READING AND WRITING CLOCK //

SUPER^.M_Execute() ;
(*//If the EMS gives the orders, the we start the process of calibration
IF IN_CmdEmsSocCalibration OR IN_CmdLocalSocCalibration THEN
	PRG_EMS.MesData.OUT_EMS.OUT_OngoingCalibration := TRUE;
	M_Calibration();
END_IF*)
END_METHOD

METHOD M_init
VAR
END_VAR
ParamPn:=2445; //apparement faudra changer la limite sur le pcs
ParamQn:=2445;
ParamSmax:=2445;
ParamSetpt_PCS_Discharge:=0.2*ParamPn;
ParamSetpt_PCS_Charge:=-0.2*ParamPn;
MesDataExd.MesCalibrationState := 0;
END_METHOD

METHOD M_Read
//////////
// Read Method for PE SKID HEMK : Modbus reading
//////////
VAR
	// Method local variables (reinitialized at each cycle) 
	MW_Float			: FB_MergeWordsToFloat;
	MW					: FB_MergeWordsToDint;
	MW_UInt				: FB_MergeWordsToUint;
	

	KK					: BYTE;						 // Index to loop over modbus blocks 	
	LL : WORD  ;
	JJ: WORD ; 
	
	CalID_AlarmPowerCol			: BYTE;
	CalIDWarning				: BYTE;
	MesSelectedDU				: WORD;
END_VAR
// CP-Read / Write 

IF MesDataExd.MesData.MesCP_Read THEN		

	// MODBUS REQUEST//
		//Electrical Measurements + Ground Measurements
		FB_ModbusRead[1]
		(
			nTCPPort		:= ParamTcpPort,
			ClockRead		:= MesDataExd.MesData.MesCP_Read AND ClockRead, 
			Reset			:= CmdClearFault_G OR IN_CmdReset_L,
			sIPAddr			:=ParamIPAddress ,
			nUnitID			:= 1, 
			tTimeout		:= ParamTimeout,
			nQuantity		:= 120 , 
			nMBAddr			:= 1000 , 
			cbLength		:= SIZEOF(MesBlock_Temp_1) , 
			pDestAddr		:= ADR(MesBlock_Temp_1) , 
			ModbusReadAlarm	=>AX_ModbusReadAlarm[1] , 
			ErrorId			=> AX_ModbusReadAlarmId[1]
		);
			
		//Production Measurements
		FB_ModbusRead[2]
		(
			nTCPPort		:= ParamTcpPort,
			ClockRead		:= MesDataExd.MesData.MesCP_Read AND ClockRead, 
			Reset			:= CmdClearFault_G OR IN_CmdReset_L,
			sIPAddr			:=ParamIPAddress , 
			nUnitID			:= 1, 
			tTimeout		:= ParamTimeout,
			nQuantity		:= 120, 
			nMBAddr			:= 1120 , 
			cbLength		:= SIZEOF(MesBlock_Temp_2) , 
			pDestAddr		:= ADR(MesBlock_Temp_2) , 
			ModbusReadAlarm	=>AX_ModbusReadAlarm[2] , 
			ErrorId			=> AX_ModbusReadAlarmId[2]
		);
	
	
	
		// DC Batterie
		FB_ModbusRead[3]
		(
			nTCPPort		:= ParamTcpPort,
			ClockRead		:= MesDataExd.MesData.MesCP_Read AND ClockRead, 
			Reset			:= CmdClearFault_G OR IN_CmdReset_L,
			sIPAddr			:=ParamIPAddress , 
			nUnitID			:= 1, 
			tTimeout		:= ParamTimeout,
			nQuantity		:= 120 , 
			nMBAddr			:= 7400 , 
			cbLength		:= SIZEOF(MesBlock_Temp_3) , 
			pDestAddr		:= ADR(MesBlock_Temp_3) , 
			ModbusReadAlarm	=>AX_ModbusReadAlarm[3] , 
			ErrorId			=> AX_ModbusReadAlarmId[3]
		);
		
		
		
	(*
		// Status Summary + Event Summary
		FB_ModbusRead[3]
		(
			nTCPPort		:= ParamTcpPort,
			ClockRead		:= MesDataExd.MesData.MesCP_Read AND ClockRead, 
			Reset			:= CmdClearFault_G OR IN_CmdReset_L,
			sIPAddr			:=ParamIPAddress , 
			nUnitID			:= 1, 
			tTimeout		:= ParamTimeout,
			nQuantity		:= 120 , 
			nMBAddr			:= 43010 , 
			cbLength		:= SIZEOF(MesBlock_Temp_3) , 
			pDestAddr		:= ADR(MesBlock_Temp_3) , 
			ModbusReadAlarm	=>AX_ModbusReadAlarm[3] , 
			ErrorId			=> AX_ModbusReadAlarmId[3]
		);
		
		*)
		
		FB_ModbusRead[4]
		(
			nTCPPort		:= ParamTcpPort,
			ClockRead		:= MesDataExd.MesData.MesCP_Read AND ClockRead, 
			Reset			:= CmdClearFault_G OR IN_CmdReset_L,
			sIPAddr			:=ParamIPAddress , 
			nUnitID			:= 1, 
			tTimeout		:= ParamTimeout,
			nQuantity		:= 100 , 
			nMBAddr			:= 1350 , 
			cbLength		:= SIZEOF(MesBlock_Temp_4)  , 
			pDestAddr		:= ADR(MesBlock_Temp_4) , 
			ModbusReadAlarm	=> AX_ModbusReadAlarm[4] , 
			ErrorId			=> AX_ModbusReadAlarmId[4]
		);
		
		FB_ModbusRead[6]
		(
			nTCPPort		:= ParamTcpPort,
			ClockRead		:= MesDataExd.MesData.MesCP_Read AND ClockRead, 
			Reset			:= CmdClearFault_G OR IN_CmdReset_L,
			sIPAddr			:=ParamIPAddress , 
			nUnitID			:= 1, 
			tTimeout		:= ParamTimeout,
			nQuantity		:= 5 , 
			nMBAddr			:= 7051 , 
			cbLength		:= SIZEOF(MesBlock_Temp_6)  , 
			pDestAddr		:= ADR(MesBlock_Temp_6) , 
			ModbusReadAlarm	=> AX_ModbusReadAlarm[6] , 
			ErrorId			=> AX_ModbusReadAlarmId[6]
		); 
		
	
		
			//Power Commands
			FOR KK:= 1 TO  ParamNbPowerCol DO 
				FB_ModbusRead_PowerCol[KK]
				(
					nTCPPort		:= ParamTcpPort,
					ClockRead		:= MesDataExd.MesData.MesCP_Read AND ClockRead, 
					Reset			:= CmdClearFault_G OR IN_CmdReset_L,
					sIPAddr			:=ParamIPAddress , 
					nUnitID			:= 1, 
					tTimeout		:= ParamTimeout,
					nQuantity		:= 32 , 
					nMBAddr			:= 5000 + 32*(KK-1) ,  
					cbLength		:= SIZEOF(MesBlock_Temp_5[KK]) , 
					pDestAddr		:= ADR(MesBlock_Temp_5[KK]) , 
					ModbusReadAlarm	=>AX_ModbusReadAlarmPowerCol[KK] , 
					ErrorId			=> AX_ModbusReadAlarmIdPowerCol[KK]
				);
		
			END_FOR
		
	
		(*
			FOR KK:= 1 TO  ParamNbDU DO 
				FB_ModbusRead_DU[KK]
				(
					nTCPPort		:= ParamTcpPort,
					ClockRead		:= MesDataExd.MesData.MesCP_Read AND ClockRead, 
					Reset			:= CmdClearFault_G OR IN_CmdReset_L,
					sIPAddr			:= ParamIPAddress , 
					nUnitID			:= 1, 
					tTimeout		:= ParamTimeout,
					nQuantity		:= 6, 
					nMBAddr			:= 45801 + 6*(KK-1),  
					cbLength		:= SIZEOF(MesBlock_Temp_6[KK]), 
					pDestAddr		:= ADR(MesBlock_Temp_6[KK]), 
					ModbusReadAlarm	=>AX_ModbusReadAlarmDU[KK], 
					ErrorId			=> AX_ModbusReadAlarmIDU[KK]
				);
		
			END_FOR
			
			*)
	
		FB_ModbusRead[7]
		(
			nTCPPort		:= ParamTcpPort,
			ClockRead		:= MesDataExd.MesData.MesCP_Read AND ClockRead, 
			Reset			:= CmdClearFault_G OR IN_CmdReset_L,
			sIPAddr			:=ParamIPAddress , 
			nUnitID			:= 1, 
			tTimeout		:= ParamTimeout,
			nQuantity		:= 10 , 
			nMBAddr			:= 5 , 
			cbLength		:= SIZEOF(MesBlock_Temp_7)  , 
			pDestAddr		:= ADR(MesBlock_Temp_7) , 
			ModbusReadAlarm	=> AX_ModbusReadAlarm[7] , 
			ErrorId			=> AX_ModbusReadAlarmId[7]
		);
		
		FB_ModbusRead[8]
		(
			nTCPPort		:= ParamTcpPort,
			ClockRead		:= MesDataExd.MesData.MesCP_Read AND ClockRead, 
			Reset			:= CmdClearFault_G OR IN_CmdReset_L,
			sIPAddr			:=ParamIPAddress , 
			nUnitID			:= 1, 
			tTimeout		:= ParamTimeout,
			nQuantity		:= 10 , 
			nMBAddr			:= 2040 , 
			cbLength		:= SIZEOF(MesBlock_Temp_8)  , 
			pDestAddr		:= ADR(MesBlock_Temp_8) , 
			ModbusReadAlarm	=> AX_ModbusReadAlarm[8] , 
			ErrorId			=> AX_ModbusReadAlarmId[8]
		);
			
			
		//test//
		MesDataExd.MesBMSSelected:=MesBlock_Temp_6[1][1];
		MesDataExd.MesSelector := MesBlock_Temp_8[1];
		
		
		MW(WORD_STRONG:= MesBlock_Temp_1[ 8], SIGNED:=TRUE, FIX:=0 , SIZE:=1, VAR_OUT:=MesDataExd.MesData.MesP);
		MW(WORD_STRONG:= MesBlock_Temp_1[ 9], SIGNED:=TRUE, FIX:=0 , SIZE:=1, VAR_OUT:=MesDataExd.MesData.MesQ);
		
		MesDataExd.MesData.MesQ:=-MesDataExd.MesData.MesQ;
		
		MW(WORD_STRONG:= MesBlock_Temp_1[ 10], SIGNED:=FALSE, FIX:=0 , SIZE:=1, VAR_OUT:=MesDataExd.MesData.MesS);
		MW(WORD_STRONG:= MesBlock_Temp_1[ 11], SIGNED:=FALSE, FIX:=3 , SIZE:=1, VAR_OUT:=MesDataExd.MesData.MesCosPhi);
		MW(WORD_STRONG:= MesBlock_Temp_1[ 12], SIGNED:=FALSE, FIX:=2 , SIZE:=1, VAR_OUT:=MesDataExd.MesData.MesFreq);	
	
		MW(WORD_STRONG:= MesBlock_Temp_1[ 31], SIGNED:=FALSE, FIX:=0 , SIZE:=1, VAR_OUT:=MesDataExd.MesU12);
		MW(WORD_STRONG:= MesBlock_Temp_1[ 32], SIGNED:=FALSE, FIX:=0 , SIZE:=1, VAR_OUT:=MesDataExd.MesU23);
		MW(WORD_STRONG:= MesBlock_Temp_1[ 33], SIGNED:=FALSE, FIX:=0 , SIZE:=1, VAR_OUT:=MesDataExd.MesU31);
		MW(WORD_STRONG:= MesBlock_Temp_1[ 34], SIGNED:=TRUE, FIX:=0 , SIZE:=1, VAR_OUT:=MesDataExd.MesI1);
		MW(WORD_STRONG:= MesBlock_Temp_1[ 35], SIGNED:=TRUE, FIX:=0 , SIZE:=1, VAR_OUT:=MesDataExd.MesI2);
		MW(WORD_STRONG:= MesBlock_Temp_1[ 36], SIGNED:=TRUE, FIX:=0 , SIZE:=1, VAR_OUT:=MesDataExd.MesI3);
	
	
		
	
		MW(WORD_STRONG:= MesBlock_Temp_1[ 51], SIGNED:=FALSE, FIX:=0 , SIZE:=1, VAR_OUT:=MesDataExd.MesData.MesUdc);  // A quoi cela correspond pour un multi psk ? 
	
		
	
		MW(WORD_STRONG:= MesBlock_Temp_1[ 61], SIGNED:=TRUE, FIX:=0 , SIZE:=1, VAR_OUT:=MesDataExd.MesData.MesPdc);
		MW(WORD_STRONG:= MesBlock_Temp_1[ 62], SIGNED:=TRUE, FIX:=0 , SIZE:=1, VAR_OUT:=MesDataExd.MesData.MesIdc);
		
		
		
		MesDataExd.MesIDState_InsuResistor_DC:=MesBlock_Temp_1[103];
		MW(WORD_STRONG:= MesBlock_Temp_1[ 104], Word_WEAK:= MesBlock_Temp_1[105], SIGNED:=FALSE, FIX:=0 , SIZE:=2, VAR_OUT:=MesDataExd.MesInsuResistor_DC);
		MesDataExd.MesIDState_InsuResistor_AC:=MesBlock_Temp_1[113];
		MW(WORD_STRONG:= MesBlock_Temp_1[ 114], Word_WEAK:= MesBlock_Temp_1[115], SIGNED:=FALSE, FIX:=0 , SIZE:=2, VAR_OUT:=MesDataExd.MesInsuResistor_AC);
		
	
		  
	
		MesDataExd.MesAlarmID:=MesBlock_Temp_2[1];
		MesDataExd.MesWarningID:=MesBlock_Temp_2[2];
		MesDataExd.MesIDState:=MesBlock_Temp_2[3];
		MW(WORD_STRONG:= MesBlock_Temp_2[ 4], SIGNED:=FALSE, FIX:=0 , SIZE:=1, VAR_OUT:=MesDataExd.MesData.MesTemp);
		MW(WORD_STRONG:= MesBlock_Temp_2[ 5], SIGNED:=FALSE, FIX:=0 , SIZE:=1, VAR_OUT:=MesDataExd.MesTemp_IGBTmax);
		MW(WORD_STRONG:= MesBlock_Temp_2[ 6], SIGNED:=FALSE, FIX:=0 , SIZE:=1, VAR_OUT:=MesDataExd.MesTemp_PowerColmax);
	
		MW(WORD_STRONG:= MesBlock_Temp_2[ 12], SIGNED:=FALSE, FIX:=0 , SIZE:=1, VAR_OUT:=MesDataExd.MesHumidity);	
		MW(WORD_STRONG:= MesBlock_Temp_2[ 21], SIGNED:=FALSE, FIX:=4 , SIZE:=1, VAR_OUT:=MesDataExd.MesPconnected);
		MW(WORD_STRONG:= MesBlock_Temp_2[ 22], SIGNED:=FALSE, FIX:=4 , SIZE:=1, VAR_OUT:=MesDataExd.MesQconnected);
	
		
		
		
		
		//MesDataExd.MesCP_Start := WORD_TO_BOOL(MesBlock_Temp_2[ 23]);
		
		//MW_REAL(WORD_STRONG:= MesBlock_Temp_2[ 58], SIGNED:=FALSE, FIX:=2 , SIZE:=1, VAR_OUT:=MesDataExd.ParamPmax); Not needed
		//MW_REAL(WORD_STRONG:= MesBlock_Temp_2[ 59], SIGNED:=FALSE, FIX:=2 , SIZE:=1, VAR_OUT:=MesDataExd.ParamQmax); Not needed
		//MW_REAL(WORD_STRONG:= MesBlock_Temp_2[ 60], SIGNED:=FALSE, FIX:=2 , SIZE:=1, VAR_OUT:=MesDataExd.ParamSmax); Not needed
		//MW(WORD_STRONG:= MesBlock_Temp_2[ 97], SIGNED:=FALSE, FIX:=0 , SIZE:=1, VAR_OUT:=MesDataExd.MesWorkingHr);
		
	
		
		
		MW(WORD_STRONG:= MesBlock_Temp_3[ 1], SIGNED:=TRUE, FIX:=0 , SIZE:=1, VAR_OUT :=MesDataExd.MesUdc_Input1);
		MW(WORD_STRONG:= MesBlock_Temp_3[ 2], SIGNED:=TRUE, FIX:=0 , SIZE:=1, VAR_OUT :=MesDataExd.MesUdc_Input2);
		MW(WORD_STRONG:= MesBlock_Temp_3[ 3], SIGNED:=TRUE, FIX:=0 , SIZE:=1, VAR_OUT :=MesDataExd.MesUdc_Input3);
		MW(WORD_STRONG:= MesBlock_Temp_3[ 4], SIGNED:=TRUE, FIX:=1 , SIZE:=1, VAR_OUT :=MesDataExd.MesUdc_Bat1);
		MW(WORD_STRONG:= MesBlock_Temp_3[ 5], SIGNED:=TRUE, FIX:=1 , SIZE:=1, VAR_OUT :=MesDataExd.MesUdc_Bat2);
		MW(WORD_STRONG:= MesBlock_Temp_3[ 6], SIGNED:=TRUE, FIX:=1 , SIZE:=1, VAR_OUT :=MesDataExd.MesUdc_Bat3);
		MW(WORD_STRONG:= MesBlock_Temp_3[ 7], SIGNED:=TRUE, FIX:=0 , SIZE:=1, VAR_OUT :=MesDataExd.MesPdc_Input1);
		MW(WORD_STRONG:= MesBlock_Temp_3[ 8], SIGNED:=TRUE, FIX:=0 , SIZE:=1, VAR_OUT :=MesDataExd.MesPdc_Input2);
		MW(WORD_STRONG:= MesBlock_Temp_3[ 9], SIGNED:=TRUE, FIX:=0 , SIZE:=1, VAR_OUT :=MesDataExd.MesPdc_Input3);
		MW(WORD_STRONG:= MesBlock_Temp_3[ 10], SIGNED:=TRUE, FIX:=0 , SIZE:=1, VAR_OUT :=MesDataExd.MesIdc_Input1);
		MW(WORD_STRONG:= MesBlock_Temp_3[ 11], SIGNED:=TRUE, FIX:=0 , SIZE:=1, VAR_OUT :=MesDataExd.MesIdc_Input2);
		MW(WORD_STRONG:= MesBlock_Temp_3[ 12], SIGNED:=TRUE, FIX:=0 , SIZE:=1, VAR_OUT :=MesDataExd.MesIdc_Input3);
		MW(WORD_STRONG:= MesBlock_Temp_3[ 17], SIGNED:=FALSE, FIX:=1 , SIZE:=1, VAR_OUT:=MesDataExd.MesIdc_RFI_Input1);
		MW(WORD_STRONG:= MesBlock_Temp_3[ 18], SIGNED:=FALSE, FIX:=1 , SIZE:=1, VAR_OUT:=MesDataExd.MesIdc_RFI_Input2);
		MW(WORD_STRONG:= MesBlock_Temp_3[ 19], SIGNED:=FALSE, FIX:=1 , SIZE:=1, VAR_OUT:=MesDataExd.MesIdc_RFI_Input3);	
		MW(WORD_STRONG:= MesBlock_Temp_3[ 32], SIGNED:=FALSE, FIX:=2 , SIZE:=1, VAR_OUT:=MesDataExd.MesP_ChargeMax);
		MW(WORD_STRONG:= MesBlock_Temp_3[ 33], SIGNED:=FALSE, FIX:=2 , SIZE:=1, VAR_OUT:=MesDataExd.MesP_DischargeMax);		
	    MW(WORD_STRONG:= MesBlock_Temp_3[ 34], SIGNED:=FALSE, FIX:=2 , SIZE:=1, VAR_OUT:=MesDataExd.MesP_ChargeMax1);
		MW(WORD_STRONG:= MesBlock_Temp_3[ 35], SIGNED:=FALSE, FIX:=2 , SIZE:=1, VAR_OUT:=MesDataExd.MesP_DischargeMax1);
		MW(WORD_STRONG:= MesBlock_Temp_3[ 36], SIGNED:=FALSE, FIX:=2 , SIZE:=1, VAR_OUT:=MesDataExd.MesP_ChargeMax2);
		MW(WORD_STRONG:= MesBlock_Temp_3[ 37], SIGNED:=FALSE, FIX:=2 , SIZE:=1, VAR_OUT:=MesDataExd.MesP_DischargeMax2);
		MW(WORD_STRONG:= MesBlock_Temp_3[ 84], Word_WEAK:= MesBlock_Temp_1[85], SIGNED:=FALSE, FIX:=0 , SIZE:=2, VAR_OUT:=MesDataExd.MesInsuResistor_DC2);
	
		MesDataExd.MesEventID := MesBlock_Temp_4[1];
		MesDataExd.MesIDState_PowerCol:=MesBlock_Temp_4[41];
		MesDataExd.MesData.MesNbPowerColConnected:=MesBlock_Temp_4[42];
	
		MesDataExd.MesReadModule 	:= MesBlock_Temp_4[101];
	
	
		
		
	// Power column/module variables 
		// Powercol[1]
	
		FOR KK:= 1 TO ParamNbPowerCol DO
			MW_UInt(WORD_STRONG:= MesBlock_Temp_5[KK][ 1], VAR_OUT := MesDataExd.AX_PowerCol[KK].MesIDState);
		
			MW(WORD_STRONG:= MesBlock_Temp_5[KK][ 2], SIGNED:=TRUE, FIX:=1 , SIZE:=1, VAR_OUT := MesDataExd.AX_PowerCol[KK].MesData.MesI1);
			MW(WORD_STRONG:= MesBlock_Temp_5[KK][ 3], SIGNED:=TRUE, FIX:=1 , SIZE:=1, VAR_OUT := MesDataExd.AX_PowerCol[KK].MesData.MesI2);
			MW(WORD_STRONG:= MesBlock_Temp_5[KK][ 4], SIGNED:=TRUE, FIX:=1 , SIZE:=1, VAR_OUT := MesDataExd.AX_PowerCol[KK].MesData.MesI3);
			MW(WORD_STRONG:= MesBlock_Temp_5[KK][ 5], SIGNED:=FALSE, FIX:=1 , SIZE:=1, VAR_OUT := MesDataExd.AX_PowerCol[KK].MesData.MesIdc);
			MW(WORD_STRONG:= MesBlock_Temp_5[KK][ 8], SIGNED:=FALSE, FIX:=0 , SIZE:=1, VAR_OUT := MesDataExd.AX_PowerCol[KK].MesData.MesUdc);
			MW(WORD_STRONG:= MesBlock_Temp_5[KK][ 9], SIGNED:=TRUE, FIX:=1 , SIZE:=1, VAR_OUT := MesDataExd.AX_PowerCol[KK].MesData.MesP);
			MW(WORD_STRONG:= MesBlock_Temp_5[KK][ 10], SIGNED:=TRUE, FIX:=1 , SIZE:=1, VAR_OUT:= MesDataExd.AX_PowerCol[KK].MesData.MesQ);
			MW(WORD_STRONG:= MesBlock_Temp_5[KK][ 11], SIGNED:=FALSE, FIX:=0 , SIZE:=1, VAR_OUT:= MesDataExd.AX_PowerCol[KK].MesData.MesTemp);
			MW(WORD_STRONG:= MesBlock_Temp_5[KK][ 12], SIGNED:=FALSE, FIX:=0 , SIZE:=1, VAR_OUT:= MesDataExd.AX_PowerCol[KK].MesTempmax);
			
			MesDataExd.AX_PowerCol[KK].MesStateIO := MesBlock_Temp_5[KK][13];
			MesDataExd.AX_PowerCol[1].MesIDState;
			MesDataExd.AX_PowerCol[2].MesIDState;
			MesDataExd.AX_PowerCol[3].MesIDState;
			MesDataExd.AX_PowerCol[4].MesIDState;
			MW(WORD_STRONG:= MesBlock_Temp_5[KK][ 32], SIGNED:=FALSE, FIX:=0 , SIZE:=1, VAR_OUT:=MesDataExd.AX_PowerCol[KK].MesHygro);
		END_FOR
		(*
			MW_UInt(WORD_STRONG:= MesBlock_Temp_3[ 1], VAR_OUT := MesDataExd.ParamID_PMode); 
			MW_UInt(WORD_STRONG:= MesBlock_Temp_3[ 2], VAR_OUT := MesDataExd.ParamID_QMode);                            
			MW(WORD_STRONG:= MesBlock_Temp_3[ 6], SIGNED:=FALSE, FIX:=3, SIZE:=1, VAR_OUT := MesDataExd.MesSetptCosPhi);
			MW(WORD_STRONG:= MesBlock_Temp_3[ 3], SIGNED:=FALSE, FIX:=2, SIZE:=1, VAR_OUT := MesDataExd.MesSetptP); 
			MW(WORD_STRONG:= MesBlock_Temp_3[ 8], SIGNED:=FALSE, FIX:=2, SIZE:=1, VAR_OUT := MesDataExd.MesSetptQ); 
		*)
	
	
	
		
		//FOR KK:= 1 TO ParamNbDU DO 
		//	IF KK <= ParamNbDU_PowerCol[1] THEN 		
		//		LL	:= 1  ;
		//		JJ	:= KK ; 
		//	ELSIF  KK <= ParamNbDU_PowerCol[1] + ParamNbDU_PowerCol[2] THEN 
		//		LL	:= 2  ;
		//		JJ	:= KK-ParamNbDU_PowerCol[1] ; 
		//	ELSE
		//		LL	:= 3  ;
		//		JJ	:= KK-ParamNbDU_PowerCol[1]-ParamNbDU_PowerCol[2] ; 			
		//	END_IF
		//// Status
		//		MesDataExd.AX_PowerCol[LL].AX_DCInputs[JJ].MesIDState := MesBlock_Temp_6[KK][4]; 
		//// Current
		//		MW(WORD_STRONG:= MesBlock_Temp_6[KK][5], SIGNED:=FALSE, FIX:=1, SIZE:=1, VAR_OUT := MesDataExd.AX_PowerCol[LL].AX_DCInputs[JJ].MesIdc); // dA ?
		//
		//// Voltage
		//	   MW(WORD_STRONG:= MesBlock_Temp_6[kk][6], SIGNED:=FALSE, FIX:=1, SIZE:=1, VAR_OUT := MesDataExd.AX_PowerCol[LL].AX_DCInputs[JJ].MesUdc); // dV ?
		//			
		//END_FOR
			
		MesDataExd.MesData.MesHeartbeat := WORD_TO_UINT(MesBlock_Temp_7[1]) MOD 2 = 0;
	
	
	
		// Evaluate 
		MesDataExd.MesData.MesI			:= (MesDataExd.MesI1 + MesDataExd.MesI2 + MesDataExd.MesI3) /3;
		MesDataExd.MesData.MesU			:= (MesDataExd.MesU12 + MesDataExd.MesU23 + MesdataExd.MesU31) /3 ; 
		
		
		
		FB_SplitWordToByte(IN:= MesDataExd.MesWarningID , STRONG_BYTE => CalID_AlarmPowerCol , WEAK_BYTE => CalIDWarning ) ; 
	
		IF CalID_AlarmPowerCol = 0 THEN 
			MesDataExd.MesWarningID :=  CalIDWarning ; 
		ELSE
			MesDataExd.AX_PowerCol[CalID_AlarmPowerCol].MesAlarmID := CalIDWarning ; 
		
		END_IF
	
		MesDataExd.MesData.MesWarning	:= MesDataExd.MesWarningID > 0 ; 
		MesDataExd.MesData.MesAlarm 	:= MesDataExd.MesAlarmID > 0 ; 
		
		MesDataExd.MesData.MesOnGrid	:= MesDataExd.MesIDState =  6 ; // ON State 
		MesDataExd.MesData.MesALOPowerCol_Connected := MesDataExd.MesData.MesNbPowerColConnected>=1 ;
		MesDataExd.MesData.MesAvailability := MesDataExd.MesPconnected*100; 
		MesDataExd.MesData.MesSnom						:= ParamSmax;	
		
		FOR KK:= 1 TO ParamNbPowerCol DO 
			MesDataExd.AX_PowerCol[KK].MesData.MesAcSwitchClosed := MesDataExd.AX_PowerCol[KK].MesStateIO.8;
			MesDataExd.AX_PowerCol[KK].MesData.MesDcSwitchClosed := MesDataExd.AX_PowerCol[KK].MesStateIO.11;
			MesDataExd.AX_PowerCol[KK].MesData.MesI :=  (MesDataExd.AX_PowerCol[KK].MesData.MesI1 + MesDataExd.AX_PowerCol[KK].MesData.MesI2 + MesDataExd.AX_PowerCol[KK].MesData.MesI3)/3 ;
		END_FOR
	 
	END_IF
END_METHOD

METHOD M_StateManager
//////////////////
// Detect which is the state of the PCS system . 
/////////////////

VAR 
	// Method local variables (reinitialized at each cycle) 
	KK :INT;
	
END_VAR
 MesDataExd.MesData.MesState 		:= 0;


IF MesDataExd.MesData.MesOpened_Ac AND  MesDataExd.MesData.MesOpened_Dc THEN 
	// OFF State :  No Charger connected or all charger in alarm
	MesDataExd.MesData.MesState.0 	:= 1 ; 
END_IF
IF MesDataExd.MesIDState = 6 OR MesDataExd.MesIDState = 10 OR MesDataExd.MesIDState = 11  THEN
	// Feeding slave
	MesDataExd.MesData.MesState.1 	:= 1 ; 

END_IF


IF MesDataExd.MesData.OUT_CmdPcsLocal THEN
	MesDataExd.MesData.MesState.2 	:= 1 ; 
END_IF


SUPER^.M_StateManager() ;
END_METHOD

METHOD M_WriteCommand
VAR
	KK : UINT;
	II : UINT;
	AX_ADR_MB			: ARRAY[1..8] OF WORD := [4251, 3009, 3199, 552, 557, 7002, 7051, 42042];
	AX_QTY_MB			: ARRAY[1..8] OF BYTE := [1, 3, 1, 1, 1, 4, 1,1];
	CmdStopRack			: BOOL;
	
	rTest : REAL := 1253;
END_VAR

// Ajust setpoint to 0 if Standby order received . 
	FB_Ramp_Standby(IN:= 0  , ASCEND := ParamPn , DESCEND := ParamPn ,TIMEBASE :=   PAramTempoStandby , RESET:= FALSE ) ; 	
	FB_Ramp_StandbyQ(IN:= 0  , ASCEND := ParamPn , DESCEND := ParamPn ,TIMEBASE :=  PAramTempoStandby , RESET:= FALSE ) ; 	

// Gestion des alarmes PCS
	// Faute batteries


(* A REPRENDRE 


	CmdInAlarmBat := AX_ESS[ParamEssNum].AX_Bat[1].MesDataExd.MesData.MesID_CmdStop_PCS = 2 OR AX_ESS[ParamEssNum].AX_Bat[2].MesDataExd.MesData.MesID_CmdStop_PCS = 2;

	F_TRIG_AlarmBat(CLK := CmdInAlarmBat);
	IF AX_ESS[ParamEssNum].AX_Bat[1].MesDataExd.MesData.MesID_CmdStop_PCS = 2 OR AX_ESS[ParamEssNum].AX_Bat[2].MesDataExd.MesData.MesID_CmdStop_PCS = 2  THEN 
		CmdStopOperation 	:= TRUE;
		MesStateFaultRack 	:= TRUE;
	END_IF	
	
	FOR KK:=1 TO CstNbBat_ESS_G DO
		FOR II:=1 TO 10 DO
			IF AX_ESS[ParamEssNum].AX_Bat[KK].MesDataExd.MesFaultString[II] > 0 THEN
				//MesStateFaultRack 	:= TRUE;
				CmdStopRack 		:= TRUE;
			END_IF
		END_FOR
	END_FOR
// Fin gestion des alarmes

*)
	
IF TP_CmdStart.Q THEN 
	bMaintainStop := FALSE ;
	FB_Ramp_Standby(RESET := TRUE , IN_RESET_VALUE := MesDataExd.MesData.MesP) ; 
	FB_Ramp_StandbyQ(RESET := TRUE , IN_RESET_VALUE :=  MesDataExd.MesData.MesQ) ; 	
ELSIF TP_CmdStandbyDelay.Q OR bMaintainStop  THEN 
	// Apply ramp at standby order 
	IN_SetptQ := FB_Ramp_StandbyQ.OUT ; 
	IN_SetptP := FB_Ramp_Standby.OUT ; 
	bMaintainStop := TRUE ;
ELSE
	FB_Ramp_Standby(RESET := TRUE , IN_RESET_VALUE := MesDataExd.MesData.MesP) ; 
	FB_Ramp_StandbyQ(RESET := TRUE , IN_RESET_VALUE :=  MesDataExd.MesData.MesQ) ; 	
END_IF

// Gestion du mode local // /

IF IN_CmdPcsInLocalMode THEN 
	IN_CmdPcsInLocalMode := FALSE;
	MesDataExd.MesData.OUT_CmdPcsLocal := NOT MesDataExd.MesData.OUT_CmdPcsLocal;
END_IF



TRIG_CmdReset	(CLK := (IN_CmdReset OR CmdClearFault_G OR IN_CmdReset) AND CalCP_Reset);
TP_Reset		(IN := TRIG_CmdReset.Q OR TRIG_CmdStart.Q, 					PT := ParamTimePulseTrig);

// delay Standby order to let time for ramp to zero
	TP_CmdStandbyDelay(IN:= IN_CmdStandby AND CalCP_Standby  , PT:= PAramTempoStandby ) ; 
	F_TRIG_Standby(CLK:= TP_CmdStandbyDelay.Q) ;
	TRIG_CmdStandby			(CLK := (F_TRIG_Standby.Q OR (TP_CmdStandbyDelay.Q AND MesDataExd.MesData.MesP < 50) ) AND NOT TP_CmdStop.Q);// Send final standby order if ramp is finished or after maximum delay
	TP_CmdStandby	(IN := TRIG_CmdStop.Q OR TRIG_CmdStandby.Q, PT := ParamTimePulseTrig);

//fault sequence
	TRIG_StandbyNow(CLK := CmdStopOperation);
	TP_CmdStandbyNow(IN := TRIG_StandbyNow.Q, PT:=T#500MS)	;
	MesAlarmsBackToNormal := (MesDataExd.MesIDState=4) AND 
	//	(AX_ESS[ParamEssNum].AX_Bat[1].MesDataExd.MesData.MesID_CmdStop_PCS = 0) AND 
	//	(AX_ESS[ParamEssNum].AX_Bat[2].MesDataExd.MesData.MesID_CmdStop_PCS = 0) AND 
		(AX_ESS[ParamEssNum].AX_Bat[1].MesDataExd.MesData.MesIDState = 3 OR AX_ESS[ParamEssNum].AX_Bat[1].MesDataExd.MesData.MesIDState = 5 ) AND
		(AX_ESS[ParamEssNum].AX_Bat[2].MesDataExd.MesData.MesIDState = 3 OR AX_ESS[ParamEssNum].AX_Bat[2].MesDataExd.MesData.MesIDState = 5 ) ;
		
	TRIG_StandbyRackEND(CLK := MesStateFaultRack  AND MesAlarmsBackToNormal);
	TP_Start(IN:=TRIG_StandbyRackEND.Q,PT:=T#500MS);
		

//Stop Sequence
	TRIG_CmdStop	(CLK := (IN_CmdStop OR IN_CmdStopOperation) AND CalCP_Stop);
	TP_CmdPreStop	(IN := TRIG_CmdStop.Q, 												PT := T#1S500MS);
	F_TrigPreStop	(CLK := TP_CmdPreStop.Q);
	TP_CmdStop		(IN := F_TrigPreStop.Q, 											PT := ParamTimePulseTrig);
	

// STart Sequence
	TRIG_CmdStart	(CLK := IN_CmdStart );  //AND CalCP_Start );
	TP_CmdPreStart	(IN := TRIG_CmdStart.Q, 											PT := ParamTimePulseTrig);
	F_TrigPreStart	(CLK := TP_CmdPreStart.Q);
	TP_CmdStart		(IN := F_TrigPreStart.Q, 											PT := ParamTimePulseTrig);



IF (IN_CmdStop OR IN_CmdStopOperation) AND CalCP_Stop THEN
	IN_CmdStop := FALSE;
END_IF

IF TRIG_CmdStart.Q THEN
	IF MesDataExd.MesData.MesAlarm THEN
		IN_CmdReset:=TRUE;
	END_IF
	FOR KK:=1 TO CstNbBat_ESS_G DO
		AX_ESS[ParamEssNum].AX_BAT[KK].IN_CmdReset := TRUE;
		AX_ESS[ParamEssNum].AX_BAT[KK].IN_CmdCloseDC := TRUE;
	END_FOR
	IN_CmdStart := FALSE;
END_IF

IF IN_CmdStandby THEN
	FOR KK:=1 TO CstNbBat_ESS_G DO
		AX_ESS[ParamEssNum].AX_BAT[KK].IN_CmdOpenDC := TRUE;
	END_FOR
	IN_CmdStandby := FALSE;
END_IF

IF  TP_CmdStandbyNow.Q THEN 
	CmdStopOperation :=FALSE;
END_IF

IF TRIG_StandbyRack.Q THEN 
	CmdStopRack :=FALSE;
END_IF

IF TRIG_StandbyRackEND.Q THEN //In case we had a Rack fault but the battey wants us to start the PCS after the standby
	MesStateFaultRack:=FALSE;
END_IF

IF IN_CmdReset  THEN
	IN_CmdReset := FALSE;
END_IF



IN_CmdWatchdog := CalLocalTimeStruct.wSecond MOD 2 = 0;
MesDataExd.OUT_CmdReset 				:= TP_Reset.Q ; 
MesDataExd.MesData.OUT_CmdStop 			:= TP_CmdStop.Q;
MesDataExd.MesData.OUT_CmdStart 		:= TP_CmdStart.Q OR TP_Start.Q;
MesDataExd.MesData.OUT_CmdStandby 		:= TP_CmdStandby.Q OR TP_CmdStandbyNow.Q OR TP_CmdStandbyRack.Q;


// Manouvers (41708)
	MesBlockWrite2_Temp[1] := BOOL_TO_WORD(MesDataExd.MesData.OUT_CmdStart );  
	MesBlockWrite2_Temp[2] := BOOL_TO_WORD(MesDataExd.MesData.OUT_CmdStandby );
	MesBlockWrite2_Temp[3] := BOOL_TO_WORD(TP_Reset.Q);


Trig_Write[1](CLK := MEMCMP(pBuf1 :=ADR(MesBlockWrite1_Temp), pBuf2 := ADR(MesBlockWrite1_Temp_Old), n := SIZEOF(MesBlockWrite1_Temp_Old))<>0);
Trig_Write[2](CLK := MEMCMP(pBuf1 :=ADR(MesBlockWrite2_Temp), pBuf2 := ADR(MesBlockWrite2_Temp_Old), n := SIZEOF(MesBlockWrite2_Temp_Old))<>0);
Trig_Write[3](CLK := MEMCMP(pBuf1 :=ADR(MesBlockWrite3_Temp), pBuf2 := ADR(MesBlockWrite3_Temp_Old), n := SIZEOF(MesBlockWrite3_Temp_Old))<>0);

